KUKA KRL program: EPS_2_25748_MH01A_A_20260121065854.src

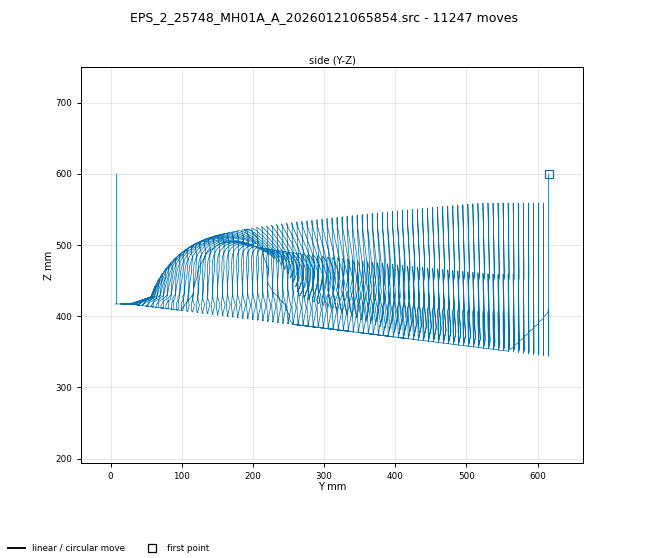
[picture p0: tool path of EPS_2_25748_MH01A_A_20260121065854.src, 11247 of 11249 moves have a stored position in this frame; points joined in program order, loops and branches not executed]
&ACCESS RVP
&REL 4
&COMMENT QRS 19112012
&PARAM EDITMASK = *
DEF PART()
EXT BAS (BAS_COMMAND :IN,REAL :IN )
INT I
BAS (#INITMOV,0 )

;KUKA QRS Post kuka4.cps  Date:22-06-2017 !

File_ID=2996

QRS_PRE_INIT()

;Init var - Until changes are made in qrs_pre_init
Outlet_Square_prg=0
Inlet_1_Square_prg=0
Inlet_2_Square_prg=0
Inlet_3_Square_prg=0
Inlet_4_Square_prg=0
Inlet_5_Square_prg=0

Outlet_1={X 0.000, Y 520.860, Z 458.500, B 0.000, E1 0.000 }
Inlet_1={X 0.000, Y 535.970, Z 408.500, B 0.000, E1 90.000 }
Outlet_1_type=201
Inlet_1_type=101
;QRS#1=Sidecore dimensions
;QRS#2=200-8" PVC SDR 35
;QRS#3=100-4" PVC SDR 28
;QRS#4=
;QRS#5=
;QRS#6=
;QRS#7=
;QRS#8=
;QRS#9=12-08 PSX
;QRS#10=8QRS PSX
;QRS#11=
;QRS#12=
;QRS#13=
;QRS#14=
;QRS#15=
;QRS#16=1220x127x838 2,75'
;QRS#17=EPS Height
;QRS#18=559
;QRS#19=*
;QRS#20= UPDATED VERSION 22-06-2017
;QRS#21=*
Outlet_Square=0100
Inlet_1_Square=045
Inlet_2_Square=0
Inlet_3_Square=0
Inlet_4_Square=0
Inlet_5_Square=0
Mill_Square=1
Outlet_Square_Prg=204
Inlet_1_Square_prg=201

QRS_INIT()

$ADVANCE=5

; T1
PTP {E1 173.434,E2 173.434}
PTP {X 0,Y 615.49,A -85,B 0,C 180,E1 173.434,E2 173.434,E3 0,E4 0,E5 0,E6 0}
QRS_SPEED_INIT()
LIN {X 0,Y 615.49,Z 600,A -85,B 0,C 180,E1 173.434,E2 173.434,E3 0,E4 0,E5 0,E6 0} C_VEL
LIN {X 0,Y 615.49,Z 432.445,A -85,B 0,C 180,E1 173.434,E2 173.434} C_VEL
LIN {X 0,Y 615.49,Z 411.751,A -85,B 0,C 180,E1 173.434,E2 173.434} C_VEL
LIN {X 0,Y 615.49,Z 411.058,A -85,B 0,C 180,E1 173.422,E2 173.422} C_VEL
LIN {X 0,Y 615.491,Z 403.195,A -85,B 0,C 180,E1 173.163,E2 173.163} C_VEL
LIN {X 0,Y 615.49,Z 396.798,A -85,B 0,C 180,E1 170.801,E2 170.801} C_VEL
LIN {X 0,Y 615.486,Z 389.623,A -85,B 0,C 180,E1 168.139,E2 168.139} C_VEL
LIN {X 0,Y 615.481,Z 382.466,A -85,B 0,C 180,E1 165.451,E2 165.451} C_VEL
LIN {X 0,Y 615.496,Z 375.278,A -85,B 0,C 180,E1 162.73,E2 162.73} C_VEL
LIN {X 0,Y 615.491,Z 368.112,A -85,B 0,C 180,E1 159.967,E2 159.967} C_VEL
LIN {X 0,Y 615.482,Z 360.924,A -85,B 0,C 180,E1 157.155,E2 157.155} C_VEL
LIN {X 0,Y 615.476,Z 354.12,A -85,B 0,C 180,E1 154.434,E2 154.434} C_VEL
LIN {X 0,Y 615.483,Z 348.349,A -85,B 0,C 180,E1 152.085,E2 152.085} C_VEL
LIN {X 0,Y 615.494,Z 343.693,A -85,B 0,C 180,E1 150.114,E2 150.114} C_VEL
LIN {X 0,Y 615.477,Z 343.693,A -85,B 0,C 180,E1 147.542,E2 147.542} C_VEL
LIN {X 0,Y 615.497,Z 343.694,A -85,B 0,C 180,E1 145.185,E2 145.185} C_VEL
LIN {X 0,Y 615.479,Z 343.69,A -85,B 0,C 180,E1 142.757,E2 142.757} C_VEL
LIN {X 0,Y 615.483,Z 343.692,A -85,B 0,C 180,E1 139.912,E2 139.912} C_VEL
LIN {X 0,Y 615.49,Z 343.699,A -85,B 0,C 180,E1 136.953,E2 136.953} C_VEL
LIN {X 0,Y 615.49,Z 343.694,A -85,B 0,C 180,E1 133.997,E2 133.997} C_VEL
LIN {X 0,Y 615.49,Z 343.689,A -85,B 0,C 180,E1 131.474,E2 131.474} C_VEL
LIN {X 0,Y 615.488,Z 343.697,A -85,B 0,C 180,E1 128.905,E2 128.905} C_VEL
LIN {X 0,Y 615.485,Z 343.69,A -85,B 0,C 180,E1 126.425,E2 126.425} C_VEL
LIN {X 0,Y 615.499,Z 343.695,A -85,B 0,C 180,E1 123.535,E2 123.535} C_VEL
LIN {X 0,Y 615.478,Z 343.692,A -85,B 0,C 180,E1 120.92,E2 120.92} C_VEL
LIN {X 0,Y 615.492,Z 343.694,A -85,B 0,C 180,E1 118.45,E2 118.45} C_VEL
LIN {X 0,Y 615.499,Z 343.694,A -85,B 0,C 180,E1 115.57,E2 115.57} C_VEL
LIN {X 0,Y 615.482,Z 343.689,A -85,B 0,C 180,E1 112.845,E2 112.845} C_VEL
LIN {X 0,Y 615.489,Z 343.693,A -85,B 0,C 180,E1 110.033,E2 110.033} C_VEL
LIN {X 0,Y 615.488,Z 343.695,A -85,B 0,C 180,E1 107.271,E2 107.271} C_VEL
LIN {X 0,Y 615.481,Z 343.69,A -85,B 0,C 180,E1 104.549,E2 104.549} C_VEL
LIN {X 0,Y 615.494,Z 343.697,A -85,B 0,C 180,E1 101.861,E2 101.861} C_VEL
LIN {X 0,Y 615.479,Z 343.692,A -85,B 0,C 180,E1 99.199,E2 99.199} C_VEL
LIN {X 0,Y 615.479,Z 343.693,A -85,B 0,C 180,E1 96.557,E2 96.557} C_VEL
LIN {X 0,Y 615.492,Z 343.694,A -85,B 0,C 180,E1 93.929,E2 93.929} C_VEL
LIN {X 0,Y 615.48,Z 343.69,A -85,B 0,C 180,E1 91.309,E2 91.309} C_VEL
LIN {X 0,Y 615.498,Z 343.7,A -85,B 0,C 180,E1 88.691,E2 88.691} C_VEL
LIN {X 0,Y 615.488,Z 343.688,A -85,B 0,C 180,E1 86.072,E2 86.072} C_VEL
LIN {X 0,Y 615.482,Z 343.697,A -85,B 0,C 180,E1 83.429,E2 83.429} C_VEL
LIN {X 0,Y 615.479,Z 343.693,A -85,B 0,C 180,E1 80.801,E2 80.801} C_VEL
LIN {X 0,Y 615.488,Z 343.69,A -85,B 0,C 180,E1 78.139,E2 78.139} C_VEL
LIN {X 0,Y 615.487,Z 343.699,A -85,B 0,C 180,E1 75.451,E2 75.451} C_VEL
LIN {X 0,Y 615.478,Z 343.691,A -85,B 0,C 180,E1 72.729,E2 72.729} C_VEL
LIN {X 0,Y 615.48,Z 343.695,A -85,B 0,C 180,E1 69.967,E2 69.967} C_VEL
LIN {X 0,Y 615.493,Z 343.696,A -85,B 0,C 180,E1 67.156,E2 67.156} C_VEL
LIN {X 0,Y 615.489,Z 343.689,A -85,B 0,C 180,E1 64.284,E2 64.284} C_VEL
LIN {X 0,Y 615.484,Z 343.69,A -85,B 0,C 180,E1 61.342,E2 61.342} C_VEL
LIN {X 0,Y 615.479,Z 343.697,A -85,B 0,C 180,E1 58.916,E2 58.916} C_VEL
LIN {X 0,Y 615.493,Z 343.69,A -85,B 0,C 180,E1 56.466,E2 56.466} C_VEL
LIN {X 0,Y 615.486,Z 343.702,A -85,B 0,C 180,E1 53.575,E2 53.575} C_VEL
LIN {X 0,Y 615.482,Z 343.69,A -85,B 0,C 180,E1 50.939,E2 50.939} C_VEL
LIN {X 0,Y 615.488,Z 343.7,A -85,B 0,C 180,E1 48.526,E2 48.526} C_VEL
LIN {X 0,Y 615.491,Z 343.689,A -85,B 0,C 180,E1 45.851,E2 45.851} C_VEL
LIN {X 0,Y 615.485,Z 343.69,A -85,B 0,C 180,E1 43.047,E2 43.047} C_VEL
LIN {X 0,Y 615.491,Z 343.693,A -85,B 0,C 180,E1 40.606,E2 40.606} C_VEL
LIN {X 0,Y 615.483,Z 343.691,A -85,B 0,C 180,E1 38.011,E2 38.011} C_VEL
LIN {X 0,Y 615.482,Z 343.694,A -85,B 0,C 180,E1 35.616,E2 35.616} C_VEL
LIN {X 0,Y 615.49,Z 343.692,A -85,B 0,C 180,E1 33.236,E2 33.236} C_VEL
LIN {X 0,Y 615.489,Z 343.688,A -85,B 0,C 180,E1 30.92,E2 30.92} C_VEL
LIN {X 0,Y 615.48,Z 343.7,A -85,B 0,C 180,E1 28.449,E2 28.449} C_VEL
LIN {X 0,Y 615.478,Z 343.693,A -85,B 0,C 180,E1 25.716,E2 25.716} C_VEL
LIN {X 0,Y 615.487,Z 343.702,A -85,B 0,C 180,E1 23.557,E2 23.557} C_VEL
LIN {X 0,Y 615.48,Z 343.692,A -85,B 0,C 180,E1 20.731,E2 20.731} C_VEL
LIN {X 0,Y 615.48,Z 343.691,A -85,B 0,C 180,E1 17.957,E2 17.957} C_VEL
LIN {X 0,Y 615.489,Z 343.702,A -85,B 0,C 180,E1 15.226,E2 15.226} C_VEL
LIN {X 0,Y 615.484,Z 343.69,A -85,B 0,C 180,E1 12.53,E2 12.53} C_VEL
LIN {X 0,Y 615.482,Z 343.694,A -85,B 0,C 180,E1 9.862,E2 9.862} C_VEL
LIN {X 0,Y 615.492,Z 343.693,A -85,B 0,C 180,E1 7.216,E2 7.216} C_VEL
LIN {X 0,Y 615.485,Z 343.69,A -85,B 0,C 180,E1 4.585,E2 4.585} C_VEL
LIN {X 0,Y 615.491,Z 343.7,A -85,B 0,C 180,E1 1.963,E2 1.963} C_VEL
LIN {X 0,Y 615.483,Z 343.689,A -85,B 0,C 180,E1 -0.654,E2 -0.654} C_VEL
LIN {X 0,Y 615.496,Z 343.696,A -85,B 0,C 180,E1 -3.273,E2 -3.273} C_VEL
LIN {X 0,Y 615.478,Z 343.692,A -85,B 0,C 180,E1 -5.899,E2 -5.899} C_VEL
LIN {X 0,Y 615.483,Z 343.693,A -85,B 0,C 180,E1 -8.537,E2 -8.537} C_VEL
LIN {X 0,Y 615.486,Z 343.695,A -85,B 0,C 180,E1 -11.193,E2 -11.193} C_VEL
LIN {X 0,Y 615.478,Z 343.69,A -85,B 0,C 180,E1 -13.928,E2 -13.928} C_VEL
LIN {X 0,Y 615.484,Z 343.7,A -85,B 0,C 180,E1 -16.587,E2 -16.587} C_VEL
LIN {X 0,Y 615.488,Z 343.691,A -85,B 0,C 180,E1 -19.338,E2 -19.338} C_VEL
LIN {X 0,Y 615.494,Z 343.687,A -85,B 0,C 180,E1 -22.136,E2 -22.136} C_VEL
LIN {X 0,Y 615.497,Z 343.695,A -85,B 0,C 180,E1 -24.991,E2 -24.991} C_VEL
LIN {X 0,Y 615.489,Z 343.688,A -85,B 0,C 180,E1 -27.177,E2 -27.177} C_VEL
LIN {X 0,Y 615.488,Z 343.693,A -85,B 0,C 180,E1 -30.16,E2 -30.16} C_VEL
LIN {X 0,Y 615.477,Z 343.691,A -85,B 0,C 180,E1 -32.458,E2 -32.458} C_VEL
LIN {X 0,Y 615.498,Z 343.7,A -85,B 0,C 180,E1 -34.815,E2 -34.815} C_VEL
LIN {X 0,Y 615.479,Z 343.69,A -85,B 0,C 180,E1 -37.243,E2 -37.243} C_VEL
LIN {X 0,Y 615.482,Z 343.696,A -85,B 0,C 180,E1 -40.088,E2 -40.088} C_VEL
LIN {X 0,Y 615.477,Z 343.69,A -85,B 0,C 180,E1 -42.354,E2 -42.354} C_VEL
LIN {X 0,Y 615.485,Z 343.696,A -85,B 0,C 180,E1 -45.069,E2 -45.069} C_VEL
LIN {X 0,Y 615.492,Z 343.694,A -85,B 0,C 180,E1 -47.92,E2 -47.92} C_VEL
LIN {X 0,Y 615.48,Z 343.694,A -85,B 0,C 180,E1 -50.249,E2 -50.249} C_VEL
LIN {X 0,Y 615.484,Z 343.7,A -85,B 0,C 180,E1 -53.064,E2 -53.064} C_VEL
LIN {X 0,Y 615.488,Z 343.691,A -85,B 0,C 180,E1 -55.3,E2 -55.3} C_VEL
LIN {X 0,Y 615.494,Z 343.689,A -85,B 0,C 180,E1 -57.669,E2 -57.669} C_VEL
LIN {X 0,Y 615.492,Z 343.687,A -85,B 0,C 180,E1 -60.594,E2 -60.594} C_VEL
LIN {X 0,Y 615.485,Z 343.84,A -85,B 0,C 180,E1 -62.593,E2 -62.593} C_VEL
LIN {X 0,Y 615.489,Z 361.437,A -85,B 0,C 180,E1 -65.369,E2 -65.369} C_VEL
LIN {X 0,Y 615.488,Z 379.893,A -85,B 0,C 180,E1 -68.216,E2 -68.216} C_VEL
LIN {X 0,Y 615.492,Z 398.328,A -85,B 0,C 180,E1 -71.009,E2 -71.009} C_VEL
LIN {X 0,Y 615.493,Z 417.271,A -85,B 0,C 180,E1 -73.832,E2 -73.832} C_VEL
LIN {X 0,Y 615.478,Z 436.291,A -85,B 0,C 180,E1 -76.631,E2 -76.631} C_VEL
LIN {X 0,Y 615.497,Z 447.778,A -85,B 0,C 180,E1 -78.306,E2 -78.306} C_VEL
LIN {X 0,Y 615.483,Z 462.241,A -85,B 0,C 180,E1 -78.557,E2 -78.557} C_VEL
LIN {X 0,Y 615.481,Z 475.314,A -85,B 0,C 180,E1 -78.921,E2 -78.921} C_VEL
LIN {X 0,Y 615.489,Z 487.118,A -85,B 0,C 180,E1 -79.383,E2 -79.383} C_VEL
LIN {X 0,Y 615.487,Z 498.575,A -85,B 0,C 180,E1 -79.972,E2 -79.972} C_VEL
LIN {X 0,Y 615.499,Z 510.021,A -85,B 0,C 180,E1 -80.719,E2 -80.719} C_VEL
LIN {X 0,Y 615.498,Z 519.257,A -85,B 0,C 180,E1 -81.464,E2 -81.464} C_VEL
LIN {X 0,Y 615.499,Z 527.654,A -85,B 0,C 180,E1 -82.29,E2 -82.29} C_VEL
LIN {X 0,Y 615.497,Z 535.69,A -85,B 0,C 180,E1 -83.259,E2 -83.259} C_VEL
LIN {X 0,Y 615.499,Z 541.423,A -85,B 0,C 180,E1 -84.102,E2 -84.102} C_VEL
LIN {X 0,Y 615.496,Z 546.873,A -85,B 0,C 180,E1 -85.087,E2 -85.087} C_VEL
LIN {X 0,Y 615.496,Z 551.141,A -85,B 0,C 180,E1 -86.072,E2 -86.072} C_VEL
LIN {X 0,Y 615.495,Z 553.399,A -85,B 0,C 180,E1 -86.727,E2 -86.727} C_VEL
LIN {X 0,Y 615.497,Z 555.233,A -85,B 0,C 180,E1 -87.382,E2 -87.382} C_VEL
LIN {X 0,Y 615.499,Z 556.608,A -85,B 0,C 180,E1 -88.037,E2 -88.037} C_VEL
LIN {X 0,Y 615.496,Z 558.174,A -85,B 0,C 180,E1 -89.346,E2 -89.346} C_VEL
LIN {X 0,Y 615.494,Z 558.389,A -85,B 0,C 180,E1 -90,E2 -90} C_VEL
LIN {X 0,Y 615.496,Z 557.58,A -85,B 0,C 180,E1 -91.309,E2 -91.309} C_VEL
LIN {X 0,Y 615.499,Z 556.607,A -85,B 0,C 180,E1 -91.963,E2 -91.963} C_VEL
LIN {X 0,Y 615.497,Z 555.233,A -85,B 0,C 180,E1 -92.618,E2 -92.618} C_VEL
LIN {X 0,Y 615.496,Z 552.349,A -85,B 0,C 180,E1 -93.601,E2 -93.601} C_VEL
LIN {X 0,Y 615.498,Z 548.441,A -85,B 0,C 180,E1 -94.585,E2 -94.585} C_VEL
LIN {X 0,Y 615.499,Z 543.404,A -85,B 0,C 180,E1 -95.57,E2 -95.57} C_VEL
LIN {X 0,Y 615.497,Z 536.869,A -85,B 0,C 180,E1 -96.583,E2 -96.583} C_VEL
LIN {X 0,Y 615.497,Z 529.132,A -85,B 0,C 180,E1 -97.545,E2 -97.545} C_VEL
LIN {X 0,Y 615.498,Z 521.044,A -85,B 0,C 180,E1 -98.371,E2 -98.371} C_VEL
LIN {X 0,Y 615.499,Z 511.166,A -85,B 0,C 180,E1 -99.199,E2 -99.199} C_VEL
LIN {X 0,Y 615.492,Z 499.979,A -85,B 0,C 180,E1 -99.945,E2 -99.945} C_VEL
LIN {X 0,Y 615.484,Z 489.021,A -85,B 0,C 180,E1 -100.527,E2 -100.527} C_VEL
LIN {X 0,Y 615.482,Z 476.474,A -85,B 0,C 180,E1 -101.041,E2 -101.041} C_VEL
LIN {X 0,Y 615.481,Z 464.062,A -85,B 0,C 180,E1 -101.402,E2 -101.402} C_VEL
LIN {X 0,Y 615.495,Z 450.456,A -85,B 0,C 180,E1 -101.652,E2 -101.652} C_VEL
LIN {X 0,Y 615.497,Z 447.777,A -85,B 0,C 180,E1 -101.694,E2 -101.694} C_VEL
LIN {X 0,Y 615.494,Z 427.093,A -85,B 0,C 180,E1 -104.718,E2 -104.718} C_VEL
LIN {X 0,Y 615.492,Z 407.537,A -85,B 0,C 180,E1 -107.613,E2 -107.613} C_VEL
LIN {X 0,Y 615.487,Z 389.681,A -85,B 0,C 180,E1 -110.295,E2 -110.295} C_VEL
LIN {X 0,Y 615.479,Z 371.82,A -85,B 0,C 180,E1 -113.023,E2 -113.023} C_VEL
LIN {X 0,Y 615.5,Z 354.513,A -85,B 0,C 180,E1 -115.715,E2 -115.715} C_VEL
LIN {X 0,Y 615.49,Z 343.697,A -85,B 0,C 180,E1 -117.453,E2 -117.453} C_VEL
LIN {X 0,Y 615.494,Z 343.698,A -85,B 0,C 180,E1 -120.16,E2 -120.16} C_VEL
LIN {X 0,Y 615.495,Z 343.696,A -85,B 0,C 180,E1 -122.457,E2 -122.457} C_VEL
LIN {X 0,Y 615.485,Z 343.698,A -85,B 0,C 180,E1 -124.815,E2 -124.815} C_VEL
LIN {X 0,Y 615.487,Z 343.701,A -85,B 0,C 180,E1 -127.242,E2 -127.242} C_VEL
LIN {X 0,Y 615.485,Z 343.698,A -85,B 0,C 180,E1 -130.088,E2 -130.088} C_VEL
LIN {X 0,Y 615.499,Z 343.696,A -85,B 0,C 180,E1 -132.352,E2 -132.352} C_VEL
LIN {X 0,Y 615.48,Z 343.699,A -85,B 0,C 180,E1 -135.07,E2 -135.07} C_VEL
LIN {X 0,Y 615.498,Z 343.7,A -85,B 0,C 180,E1 -137.919,E2 -137.919} C_VEL
LIN {X 0,Y 615.492,Z 343.697,A -85,B 0,C 180,E1 -140.25,E2 -140.25} C_VEL
LIN {X 0,Y 615.485,Z 343.702,A -85,B 0,C 180,E1 -143.064,E2 -143.064} C_VEL
LIN {X 0,Y 615.491,Z 343.697,A -85,B 0,C 180,E1 -145.978,E2 -145.978} C_VEL
LIN {X 0,Y 615.496,Z 343.699,A -85,B 0,C 180,E1 -148.315,E2 -148.315} C_VEL
LIN {X 0,Y 615.491,Z 343.791,A -85,B 0,C 180,E1 -150.303,E2 -150.303} C_VEL
LIN {X 0,Y 615.498,Z 350.25,A -85,B 0,C 180,E1 -152.954,E2 -152.954} C_VEL
LIN {X 0,Y 615.489,Z 357.77,A -85,B 0,C 180,E1 -155.992,E2 -155.992} C_VEL
LIN {X 0,Y 615.478,Z 364.291,A -85,B 0,C 180,E1 -158.568,E2 -158.568} C_VEL
LIN {X 0,Y 615.477,Z 371.461,A -85,B 0,C 180,E1 -161.354,E2 -161.354} C_VEL
LIN {X 0,Y 615.492,Z 378.634,A -85,B 0,C 180,E1 -164.095,E2 -164.095} C_VEL
LIN {X 0,Y 615.494,Z 385.799,A -85,B 0,C 180,E1 -166.799,E2 -166.799} C_VEL
LIN {X 0,Y 615.486,Z 392.972,A -85,B 0,C 180,E1 -169.473,E2 -169.473} C_VEL
LIN {X 0,Y 615.477,Z 400.129,A -85,B 0,C 180,E1 -172.124,E2 -172.124} C_VEL
LIN {X 0,Y 615.484,Z 403.219,A -85,B 0,C 180,E1 -173.261,E2 -173.261} C_VEL
LIN {X 0,Y 615.493,Z 413.526,A -85,B 0,C 180,E1 -173.608,E2 -173.608} C_VEL
LIN {X 0,Y 615.478,Z 421.946,A -85,B 0,C 180,E1 -174.019,E2 -174.019} C_VEL
LIN {X 0,Y 615.486,Z 429.671,A -85,B 0,C 180,E1 -174.512,E2 -174.512} C_VEL
LIN {X 0,Y 615.481,Z 436.518,A -85,B 0,C 180,E1 -175.087,E2 -175.087} C_VEL
LIN {X 0,Y 615.497,Z 442.668,A -85,B 0,C 180,E1 -175.744,E2 -175.744} C_VEL
LIN {X 0,Y 615.497,Z 447.515,A -85,B 0,C 180,E1 -176.399,E2 -176.399} C_VEL
LIN {X 0,Y 615.496,Z 451.25,A -85,B 0,C 180,E1 -177.055,E2 -177.055} C_VEL
LIN {X 0,Y 615.498,Z 455.23,A -85,B 0,C 180,E1 -178.037,E2 -178.037} C_VEL
LIN {X 0,Y 615.495,Z 456.964,A -85,B 0,C 180,E1 -178.691,E2 -178.691} C_VEL
LIN {X 0,Y 615.497,Z 458.004,A -85,B 0,C 180,E1 -179.346,E2 -179.346} C_VEL
LIN {X 0,Y 615.494,Z 458.384,A -85,B 0,C 180,E1 -180,E2 -180} C_VEL
LIN {X 0,Y 615.496,Z 458.105,A -85,B 0,C 180,E1 -180.654,E2 -180.654} C_VEL
LIN {X 0,Y 615.498,Z 457.165,A -85,B 0,C 180,E1 -181.309,E2 -181.309} C_VEL
LIN {X 0,Y 615.496,Z 455.536,A -85,B 0,C 180,E1 -181.963,E2 -181.963} C_VEL
LIN {X 0,Y 615.498,Z 451.663,A -85,B 0,C 180,E1 -182.945,E2 -182.945} C_VEL
LIN {X 0,Y 615.5,Z 447.011,A -85,B 0,C 180,E1 -183.765,E2 -183.765} C_VEL
LIN {X 0,Y 615.499,Z 442.03,A -85,B 0,C 180,E1 -184.42,E2 -184.42} C_VEL
LIN {X 0,Y 615.492,Z 435.752,A -85,B 0,C 180,E1 -185.077,E2 -185.077} C_VEL
LIN {X 0,Y 615.483,Z 428.588,A -85,B 0,C 180,E1 -185.652,E2 -185.652} C_VEL
LIN {X 0,Y 615.483,Z 420.604,A -85,B 0,C 180,E1 -186.145,E2 -186.145} C_VEL
LIN {X 0,Y 615.49,Z 411.058,A -85,B 0,C 180,E1 -186.578,E2 -186.578} C_VEL
LIN {X 0,Y 615.134,Z 407.804,A -85,B 0,C 180,E1 -186.754,E2 -186.754} C_VEL
LIN {X 0,Y 614.28,Z 405.203,A -85,B 0,C 180,E1 -187.003,E2 -187.003} C_VEL
LIN {X 0,Y 612.526,Z 402.365,A -85,B 0,C 180,E1 -187.458,E2 -187.458} C_VEL
LIN {X 0,Y 610.614,Z 400.714,A -85,B 0,C 180,E1 -187.986,E2 -187.986} C_VEL
LIN {X 0,Y 608.705,Z 398.756,A -85,B 0,C 180,E1 -188.746,E2 -188.746} C_VEL
LIN {X 0,Y 608.412,Z 397.698,A -85,B 0,C 180,E1 -189.134,E2 -189.134} C_VEL
LIN {X 0,Y 608.424,Z 390.014,A -85,B 0,C 180,E1 -192.001,E2 -192.001} C_VEL
LIN {X 0,Y 608.441,Z 382.795,A -85,B 0,C 180,E1 -194.721,E2 -194.721} C_VEL
LIN {X 0,Y 608.459,Z 375.575,A -85,B 0,C 180,E1 -197.477,E2 -197.477} C_VEL
LIN {X 0,Y 608.443,Z 368.356,A -85,B 0,C 180,E1 -200.275,E2 -200.275} C_VEL
LIN {X 0,Y 608.446,Z 361.136,A -85,B 0,C 180,E1 -203.124,E2 -203.124} C_VEL
LIN {X 0,Y 608.465,Z 354.69,A -85,B 0,C 180,E1 -205.719,E2 -205.719} C_VEL
LIN {X 0,Y 608.476,Z 347.645,A -85,B 0,C 180,E1 -208.62,E2 -208.62} C_VEL
LIN {X 0,Y 608.481,Z 344.69,A -85,B 0,C 180,E1 -209.905,E2 -209.905} C_VEL
LIN {X 0,Y 608.454,Z 344.692,A -85,B 0,C 180,E1 -212.521,E2 -212.521} C_VEL
LIN {X 0,Y 608.444,Z 344.692,A -85,B 0,C 180,E1 -215.278,E2 -215.278} C_VEL
LIN {X 0,Y 608.468,Z 344.693,A -85,B 0,C 180,E1 -217.747,E2 -217.747} C_VEL
LIN {X 0,Y 608.448,Z 344.691,A -85,B 0,C 180,E1 -220.328,E2 -220.328} C_VEL
LIN {X 0,Y 608.455,Z 344.698,A -85,B 0,C 180,E1 -222.96,E2 -222.96} C_VEL
LIN {X 0,Y 608.461,Z 344.69,A -85,B 0,C 180,E1 -225.736,E2 -225.736} C_VEL
LIN {X 0,Y 608.464,Z 344.689,A -85,B 0,C 180,E1 -228.658,E2 -228.658} C_VEL
LIN {X 0,Y 608.465,Z 344.69,A -85,B 0,C 180,E1 -231.76,E2 -231.76} C_VEL
LIN {X 0,Y 608.448,Z 344.691,A -85,B 0,C 180,E1 -233.955,E2 -233.955} C_VEL
LIN {X 0,Y 608.47,Z 344.696,A -85,B 0,C 180,E1 -236.329,E2 -236.329} C_VEL
LIN {X 0,Y 608.449,Z 344.691,A -85,B 0,C 180,E1 -238.733,E2 -238.733} C_VEL
LIN {X 0,Y 608.479,Z 344.694,A -85,B 0,C 180,E1 -241.38,E2 -241.38} C_VEL
LIN {X 0,Y 608.446,Z 344.692,A -85,B 0,C 180,E1 -243.964,E2 -243.964} C_VEL
LIN {X 0,Y 608.465,Z 344.694,A -85,B 0,C 180,E1 -246.155,E2 -246.155} C_VEL
LIN {X 0,Y 608.47,Z 344.691,A -85,B 0,C 180,E1 -248.308,E2 -248.308} C_VEL
LIN {X 0,Y 608.457,Z 344.695,A -85,B 0,C 180,E1 -251.13,E2 -251.13} C_VEL
LIN {X 0,Y 608.459,Z 344.69,A -85,B 0,C 180,E1 -253.906,E2 -253.906} C_VEL
LIN {X 0,Y 608.46,Z 344.693,A -85,B 0,C 180,E1 -256.643,E2 -256.643} C_VEL
LIN {X 0,Y 608.466,Z 344.692,A -85,B 0,C 180,E1 -259.35,E2 -259.35} C_VEL
LIN {X 0,Y 608.481,Z 344.687,A -85,B 0,C 180,E1 -262.033,E2 -262.033} C_VEL
LIN {X 0,Y 608.472,Z 344.695,A -85,B 0,C 180,E1 -264.698,E2 -264.698} C_VEL
LIN {X 0,Y 608.472,Z 344.688,A -85,B 0,C 180,E1 -267.352,E2 -267.352} C_VEL
LIN {X 0,Y 608.482,Z 344.69,A -85,B 0,C 180,E1 -270,E2 -270} C_VEL
LIN {X 0,Y 608.472,Z 344.691,A -85,B 0,C 180,E1 -272.648,E2 -272.648} C_VEL
LIN {X 0,Y 608.462,Z 344.69,A -85,B 0,C 180,E1 -275.302,E2 -275.302} C_VEL
LIN {X 0,Y 608.482,Z 344.694,A -85,B 0,C 180,E1 -277.967,E2 -277.967} C_VEL
LIN {X 0,Y 608.47,Z 344.691,A -85,B 0,C 180,E1 -280.954,E2 -280.954} C_VEL
LIN {X 0,Y 608.465,Z 344.692,A -85,B 0,C 180,E1 -283.356,E2 -283.356} C_VEL
LIN {X 0,Y 608.468,Z 344.692,A -85,B 0,C 180,E1 -286.094,E2 -286.094} C_VEL
LIN {X 0,Y 608.457,Z 344.69,A -85,B 0,C 180,E1 -288.87,E2 -288.87} C_VEL
LIN {X 0,Y 608.472,Z 344.691,A -85,B 0,C 180,E1 -291.691,E2 -291.691} C_VEL
LIN {X 0,Y 608.451,Z 344.697,A -85,B 0,C 180,E1 -294.571,E2 -294.571} C_VEL
LIN {X 0,Y 608.472,Z 344.688,A -85,B 0,C 180,E1 -297.205,E2 -297.205} C_VEL
LIN {X 0,Y 608.465,Z 344.693,A -85,B 0,C 180,E1 -299.971,E2 -299.971} C_VEL
LIN {X 0,Y 608.464,Z 344.694,A -85,B 0,C 180,E1 -302.879,E2 -302.879} C_VEL
LIN {X 0,Y 608.446,Z 344.692,A -85,B 0,C 180,E1 -305.278,E2 -305.278} C_VEL
LIN {X 0,Y 608.472,Z 344.693,A -85,B 0,C 180,E1 -308.24,E2 -308.24} C_VEL
LIN {X 0,Y 608.447,Z 344.692,A -85,B 0,C 180,E1 -310.328,E2 -310.328} C_VEL
LIN {X 0,Y 608.485,Z 344.69,A -85,B 0,C 180,E1 -313.31,E2 -313.31} C_VEL
LIN {X 0,Y 608.469,Z 344.692,A -85,B 0,C 180,E1 -316.13,E2 -316.13} C_VEL
LIN {X 0,Y 608.451,Z 344.691,A -85,B 0,C 180,E1 -318.823,E2 -318.823} C_VEL
LIN {X 0,Y 608.465,Z 344.691,A -85,B 0,C 180,E1 -321.76,E2 -321.76} C_VEL
LIN {X 0,Y 608.451,Z 344.691,A -85,B 0,C 180,E1 -323.954,E2 -323.954} C_VEL
LIN {X 0,Y 608.471,Z 344.695,A -85,B 0,C 180,E1 -326.329,E2 -326.329} C_VEL
LIN {X 0,Y 608.449,Z 344.691,A -85,B 0,C 180,E1 -328.732,E2 -328.732} C_VEL
LIN {X 0,Y 608.472,Z 344.695,A -85,B 0,C 180,E1 -331.381,E2 -331.381} C_VEL
LIN {X 0,Y 608.437,Z 344.692,A -85,B 0,C 180,E1 -333.964,E2 -333.964} C_VEL
LIN {X 0,Y 608.471,Z 344.692,A -85,B 0,C 180,E1 -336.155,E2 -336.155} C_VEL
LIN {X 0,Y 608.454,Z 344.69,A -85,B 0,C 180,E1 -339.018,E2 -339.018} C_VEL
LIN {X 0,Y 608.448,Z 344.693,A -85,B 0,C 180,E1 -341.828,E2 -341.828} C_VEL
LIN {X 0,Y 608.471,Z 344.693,A -85,B 0,C 180,E1 -344.594,E2 -344.594} C_VEL
LIN {X 0,Y 608.476,Z 344.688,A -85,B 0,C 180,E1 -347.323,E2 -347.323} C_VEL
LIN {X 0,Y 608.453,Z 344.694,A -85,B 0,C 180,E1 -350.023,E2 -350.023} C_VEL
LIN {X 0,Y 608.469,Z 344.691,A -85,B 0,C 180,E1 -352.701,E2 -352.701} C_VEL
LIN {X 0,Y 608.455,Z 344.691,A -85,B 0,C 180,E1 -355.362,E2 -355.362} C_VEL
LIN {X 0,Y 608.46,Z 344.696,A -85,B 0,C 180,E1 -358.014,E2 -358.014} C_VEL
LIN {X 0,Y 608.478,Z 344.687,A -85,B 0,C 180,E1 -360.662,E2 -360.662} C_VEL
LIN {X 0,Y 608.488,Z 344.691,A -85,B 0,C 180,E1 -363.311,E2 -363.311} C_VEL
LIN {X 0,Y 608.453,Z 344.692,A -85,B 0,C 180,E1 -365.967,E2 -365.967} C_VEL
LIN {X 0,Y 608.455,Z 344.691,A -85,B 0,C 180,E1 -368.636,E2 -368.636} C_VEL
LIN {X 0,Y 608.477,Z 344.693,A -85,B 0,C 180,E1 -371.324,E2 -371.324} C_VEL
LIN {X 0,Y 608.471,Z 344.688,A -85,B 0,C 180,E1 -374.037,E2 -374.037} C_VEL
LIN {X 0,Y 608.477,Z 344.69,A -85,B 0,C 180,E1 -376.783,E2 -376.783} C_VEL
LIN {X 0,Y 608.457,Z 344.694,A -85,B 0,C 180,E1 -379.57,E2 -379.57} C_VEL
LIN {X 0,Y 608.462,Z 344.69,A -85,B 0,C 180,E1 -382.476,E2 -382.476} C_VEL
LIN {X 0,Y 608.46,Z 344.694,A -85,B 0,C 180,E1 -384.571,E2 -384.571} C_VEL
LIN {X 0,Y 608.452,Z 344.691,A -85,B 0,C 180,E1 -387.518,E2 -387.518} C_VEL
LIN {X 0,Y 608.475,Z 344.693,A -85,B 0,C 180,E1 -389.972,E2 -389.972} C_VEL
LIN {X 0,Y 608.457,Z 344.694,A -85,B 0,C 180,E1 -392.88,E2 -392.88} C_VEL
LIN {X 0,Y 608.445,Z 344.693,A -85,B 0,C 180,E1 -395.278,E2 -395.278} C_VEL
LIN {X 0,Y 608.476,Z 344.694,A -85,B 0,C 180,E1 -398.241,E2 -398.241} C_VEL
LIN {X 0,Y 608.453,Z 344.693,A -85,B 0,C 180,E1 -401.177,E2 -401.177} C_VEL
LIN {X 0,Y 608.47,Z 344.688,A -85,B 0,C 180,E1 -403.87,E2 -403.87} C_VEL
LIN {X 0,Y 608.483,Z 344.691,A -85,B 0,C 180,E1 -406.69,E2 -406.69} C_VEL
LIN {X 0,Y 608.455,Z 344.691,A -85,B 0,C 180,E1 -408.823,E2 -408.823} C_VEL
LIN {X 0,Y 608.464,Z 344.693,A -85,B 0,C 180,E1 -411.76,E2 -411.76} C_VEL
LIN {X 0,Y 608.447,Z 344.691,A -85,B 0,C 180,E1 -413.955,E2 -413.955} C_VEL
LIN {X 0,Y 608.468,Z 344.693,A -85,B 0,C 180,E1 -416.329,E2 -416.329} C_VEL
LIN {X 0,Y 608.448,Z 344.692,A -85,B 0,C 180,E1 -418.733,E2 -418.733} C_VEL
LIN {X 0,Y 608.474,Z 344.694,A -85,B 0,C 180,E1 -421.38,E2 -421.38} C_VEL
LIN {X 0,Y 608.479,Z 344.706,A -85,B 0,C 180,E1 -422.39,E2 -422.39} C_VEL
LIN {X 0,Y 608.617,Z 357.707,A -85,B 0,C 180,E1 -424.481,E2 -424.481} C_VEL
LIN {X 0,Y 608.571,Z 375.515,A -85,B 0,C 180,E1 -427.276,E2 -427.276} C_VEL
LIN {X 0,Y 608.516,Z 393.747,A -85,B 0,C 180,E1 -430.08,E2 -430.08} C_VEL
LIN {X 0,Y 608.5,Z 411.056,A -85,B 0,C 180,E1 -432.698,E2 -432.698} C_VEL
LIN {X 0,Y 608.47,Z 429.518,A -85,B 0,C 180,E1 -435.45,E2 -435.45} C_VEL
LIN {X 0,Y 608.486,Z 447.981,A -85,B 0,C 180,E1 -438.17,E2 -438.17} C_VEL
LIN {X 0,Y 608.545,Z 463.267,A -85,B 0,C 180,E1 -438.445,E2 -438.445} C_VEL
LIN {X 0,Y 608.523,Z 475.887,A -85,B 0,C 180,E1 -438.808,E2 -438.808} C_VEL
LIN {X 0,Y 608.519,Z 487.581,A -85,B 0,C 180,E1 -439.275,E2 -439.275} C_VEL
LIN {X 0,Y 608.492,Z 498.755,A -85,B 0,C 180,E1 -439.855,E2 -439.855} C_VEL
LIN {X 0,Y 608.504,Z 510.252,A -85,B 0,C 180,E1 -440.611,E2 -440.611} C_VEL
LIN {X 0,Y 608.472,Z 519.536,A -85,B 0,C 180,E1 -441.364,E2 -441.364} C_VEL
LIN {X 0,Y 608.456,Z 527.989,A -85,B 0,C 180,E1 -442.2,E2 -442.2} C_VEL
LIN {X 0,Y 608.462,Z 536.235,A -85,B 0,C 180,E1 -443.201,E2 -443.201} C_VEL
LIN {X 0,Y 608.437,Z 542.877,A -85,B 0,C 180,E1 -444.199,E2 -444.199} C_VEL
LIN {X 0,Y 608.432,Z 548.95,A -85,B 0,C 180,E1 -445.362,E2 -445.362} C_VEL
LIN {X 0,Y 608.449,Z 552.896,A -85,B 0,C 180,E1 -446.358,E2 -446.358} C_VEL
LIN {X 0,Y 608.425,Z 555.809,A -85,B 0,C 180,E1 -447.352,E2 -447.352} C_VEL
LIN {X 0,Y 608.444,Z 557.201,A -85,B 0,C 180,E1 -448.014,E2 -448.014} C_VEL
LIN {X 0,Y 608.438,Z 558.783,A -85,B 0,C 180,E1 -449.338,E2 -449.338} C_VEL
LIN {X 0,Y 608.434,Z 559,A -85,B 0,C 180,E1 -450,E2 -450} C_VEL
LIN {X 0,Y 608.448,Z 558.184,A -85,B 0,C 180,E1 -451.324,E2 -451.324} C_VEL
LIN {X 0,Y 608.444,Z 557.201,A -85,B 0,C 180,E1 -451.986,E2 -451.986} C_VEL
LIN {X 0,Y 608.425,Z 555.809,A -85,B 0,C 180,E1 -452.648,E2 -452.648} C_VEL
LIN {X 0,Y 608.449,Z 552.896,A -85,B 0,C 180,E1 -453.642,E2 -453.642} C_VEL
LIN {X 0,Y 608.432,Z 548.95,A -85,B 0,C 180,E1 -454.638,E2 -454.638} C_VEL
LIN {X 0,Y 608.437,Z 542.876,A -85,B 0,C 180,E1 -455.801,E2 -455.801} C_VEL
LIN {X 0,Y 608.462,Z 536.234,A -85,B 0,C 180,E1 -456.799,E2 -456.799} C_VEL
LIN {X 0,Y 608.456,Z 527.988,A -85,B 0,C 180,E1 -457.8,E2 -457.8} C_VEL
LIN {X 0,Y 608.472,Z 519.535,A -85,B 0,C 180,E1 -458.636,E2 -458.636} C_VEL
LIN {X 0,Y 608.481,Z 509.089,A -85,B 0,C 180,E1 -459.473,E2 -459.473} C_VEL
LIN {X 0,Y 608.492,Z 498.754,A -85,B 0,C 180,E1 -460.145,E2 -460.145} C_VEL
LIN {X 0,Y 608.521,Z 487.26,A -85,B 0,C 180,E1 -460.74,E2 -460.74} C_VEL
LIN {X 0,Y 608.529,Z 474.882,A -85,B 0,C 180,E1 -461.225,E2 -461.225} C_VEL
LIN {X 0,Y 608.546,Z 461.434,A -85,B 0,C 180,E1 -461.597,E2 -461.597} C_VEL
LIN {X 0,Y 608.486,Z 447.98,A -85,B 0,C 180,E1 -461.83,E2 -461.83} C_VEL
LIN {X 0,Y 608.49,Z 428.364,A -85,B 0,C 180,E1 -464.72,E2 -464.72} C_VEL
LIN {X 0,Y 608.502,Z 409.901,A -85,B 0,C 180,E1 -467.475,E2 -467.475} C_VEL
LIN {X 0,Y 608.531,Z 392.592,A -85,B 0,C 180,E1 -470.096,E2 -470.096} C_VEL
LIN {X 0,Y 608.572,Z 374.131,A -85,B 0,C 180,E1 -472.939,E2 -472.939} C_VEL
LIN {X 0,Y 608.614,Z 356.269,A -85,B 0,C 180,E1 -475.748,E2 -475.748} C_VEL
LIN {X 0,Y 608.483,Z 344.705,A -85,B 0,C 180,E1 -477.61,E2 -477.61} C_VEL
LIN {X 0,Y 608.477,Z 344.692,A -85,B 0,C 180,E1 -480.545,E2 -480.545} C_VEL
LIN {X 0,Y 608.465,Z 344.695,A -85,B 0,C 180,E1 -482.879,E2 -482.879} C_VEL
LIN {X 0,Y 608.443,Z 344.699,A -85,B 0,C 180,E1 -485.278,E2 -485.278} C_VEL
LIN {X 0,Y 608.466,Z 344.694,A -85,B 0,C 180,E1 -487.747,E2 -487.747} C_VEL
LIN {X 0,Y 608.453,Z 344.697,A -85,B 0,C 180,E1 -490.329,E2 -490.329} C_VEL
LIN {X 0,Y 608.483,Z 344.692,A -85,B 0,C 180,E1 -493.31,E2 -493.31} C_VEL
LIN {X 0,Y 608.479,Z 344.692,A -85,B 0,C 180,E1 -496.131,E2 -496.131} C_VEL
LIN {X 0,Y 608.457,Z 344.697,A -85,B 0,C 180,E1 -498.823,E2 -498.823} C_VEL
LIN {X 0,Y 608.474,Z 344.693,A -85,B 0,C 180,E1 -501.412,E2 -501.412} C_VEL
LIN {X 0,Y 608.465,Z 344.695,A -85,B 0,C 180,E1 -503.953,E2 -503.953} C_VEL
LIN {X 0,Y 608.469,Z 344.696,A -85,B 0,C 180,E1 -506.33,E2 -506.33} C_VEL
LIN {X 0,Y 608.45,Z 344.696,A -85,B 0,C 180,E1 -508.732,E2 -508.732} C_VEL
LIN {X 0,Y 608.483,Z 344.805,A -85,B 0,C 180,E1 -510.316,E2 -510.316} C_VEL
LIN {X 0,Y 608.451,Z 351.891,A -85,B 0,C 180,E1 -513.226,E2 -513.226} C_VEL
LIN {X 0,Y 608.458,Z 358.354,A -85,B 0,C 180,E1 -515.852,E2 -515.852} C_VEL
LIN {X 0,Y 608.443,Z 364.518,A -85,B 0,C 180,E1 -518.307,E2 -518.307} C_VEL
LIN {X 0,Y 608.432,Z 371.734,A -85,B 0,C 180,E1 -521.13,E2 -521.13} C_VEL
LIN {X 0,Y 608.448,Z 378.95,A -85,B 0,C 180,E1 -523.906,E2 -523.906} C_VEL
LIN {X 0,Y 608.437,Z 386.166,A -85,B 0,C 180,E1 -526.643,E2 -526.643} C_VEL
LIN {X 0,Y 608.424,Z 393.383,A -85,B 0,C 180,E1 -529.349,E2 -529.349} C_VEL
LIN {X 0,Y 608.412,Z 400.599,A -85,B 0,C 180,E1 -532.032,E2 -532.032} C_VEL
LIN {X 0,Y 608.446,Z 403.882,A -85,B 0,C 180,E1 -533.187,E2 -533.187} C_VEL
LIN {X 0,Y 608.478,Z 414.08,A -85,B 0,C 180,E1 -533.534,E2 -533.534} C_VEL
LIN {X 0,Y 608.454,Z 422.473,A -85,B 0,C 180,E1 -533.95,E2 -533.95} C_VEL
LIN {X 0,Y 608.451,Z 431.253,A -85,B 0,C 180,E1 -534.532,E2 -534.532} C_VEL
LIN {X 0,Y 608.44,Z 437.028,A -85,B 0,C 180,E1 -535.03,E2 -535.03} C_VEL
LIN {X 0,Y 608.443,Z 443.206,A -85,B 0,C 180,E1 -535.694,E2 -535.694} C_VEL
LIN {X 0,Y 608.451,Z 448.068,A -85,B 0,C 180,E1 -536.358,E2 -536.358} C_VEL
LIN {X 0,Y 608.451,Z 451.818,A -85,B 0,C 180,E1 -537.021,E2 -537.021} C_VEL
LIN {X 0,Y 608.443,Z 455.825,A -85,B 0,C 180,E1 -538.014,E2 -538.014} C_VEL
LIN {X 0,Y 608.448,Z 457.569,A -85,B 0,C 180,E1 -538.676,E2 -538.676} C_VEL
LIN {X 0,Y 608.44,Z 458.615,A -85,B 0,C 180,E1 -539.338,E2 -539.338} C_VEL
LIN {X 0,Y 608.434,Z 458.995,A -85,B 0,C 180,E1 -540,E2 -540} C_VEL
LIN {X 0,Y 608.438,Z 458.714,A -85,B 0,C 180,E1 -540.662,E2 -540.662} C_VEL
LIN {X 0,Y 608.45,Z 457.768,A -85,B 0,C 180,E1 -541.324,E2 -541.324} C_VEL
LIN {X 0,Y 608.442,Z 456.128,A -85,B 0,C 180,E1 -541.986,E2 -541.986} C_VEL
LIN {X 0,Y 608.429,Z 453.745,A -85,B 0,C 180,E1 -542.648,E2 -542.648} C_VEL
LIN {X 0,Y 608.452,Z 448.617,A -85,B 0,C 180,E1 -543.642,E2 -543.642} C_VEL
LIN {X 0,Y 608.452,Z 442.554,A -85,B 0,C 180,E1 -544.472,E2 -544.472} C_VEL
LIN {X 0,Y 608.442,Z 436.249,A -85,B 0,C 180,E1 -545.136,E2 -545.136} C_VEL
LIN {X 0,Y 608.458,Z 429.092,A -85,B 0,C 180,E1 -545.718,E2 -545.718} C_VEL
LIN {X 0,Y 608.443,Z 421.106,A -85,B 0,C 180,E1 -546.217,E2 -546.217} C_VEL
LIN {X 0,Y 608.478,Z 411.444,A -85,B 0,C 180,E1 -546.661,E2 -546.661} C_VEL
LIN {X 0,Y 608.431,Z 403.701,A -85,B 0,C 180,E1 -546.91,E2 -546.91} C_VEL
LIN {X 0,Y 608.412,Z 397.698,A -85,B 0,C 180,E1 -549.134,E2 -549.134} C_VEL
LIN {X 0,Y 607.751,Z 396.282,A -85,B 0,C 180,E1 -549.671,E2 -549.671} C_VEL
LIN {X 0,Y 604.862,Z 394.078,A -85,B 0,C 180,E1 -550.543,E2 -550.543} C_VEL
LIN {X 0,Y 602.428,Z 392.33,A -85,B 0,C 180,E1 -551.245,E2 -551.245} C_VEL
LIN {X 0,Y 601.405,Z 390.951,A -85,B 0,C 180,E1 -551.787,E2 -551.787} C_VEL
LIN {X 0,Y 601.333,Z 390.473,A -85,B 0,C 180,E1 -551.97,E2 -551.97} C_VEL
LIN {X 0,Y 601.361,Z 382.793,A -85,B 0,C 180,E1 -554.899,E2 -554.899} C_VEL
LIN {X 0,Y 601.377,Z 375.574,A -85,B 0,C 180,E1 -557.689,E2 -557.689} C_VEL
LIN {X 0,Y 601.367,Z 368.354,A -85,B 0,C 180,E1 -560.524,E2 -560.524} C_VEL
LIN {X 0,Y 601.38,Z 361.134,A -85,B 0,C 180,E1 -563.412,E2 -563.412} C_VEL
LIN {X 0,Y 601.395,Z 355.127,A -85,B 0,C 180,E1 -565.863,E2 -565.863} C_VEL
LIN {X 0,Y 601.435,Z 348.094,A -85,B 0,C 180,E1 -568.788,E2 -568.788} C_VEL
LIN {X 0,Y 601.423,Z 345.57,A -85,B 0,C 180,E1 -569.865,E2 -569.865} C_VEL
LIN {X 0,Y 601.417,Z 345.571,A -85,B 0,C 180,E1 -572.714,E2 -572.714} C_VEL
LIN {X 0,Y 601.403,Z 345.57,A -85,B 0,C 180,E1 -575.113,E2 -575.113} C_VEL
LIN {X 0,Y 601.437,Z 345.566,A -85,B 0,C 180,E1 -577.419,E2 -577.419} C_VEL
LIN {X 0,Y 601.416,Z 345.569,A -85,B 0,C 180,E1 -579.995,E2 -579.995} C_VEL
LIN {X 0,Y 601.412,Z 345.571,A -85,B 0,C 180,E1 -582.671,E2 -582.671} C_VEL
LIN {X 0,Y 601.431,Z 345.565,A -85,B 0,C 180,E1 -585.482,E2 -585.482} C_VEL
LIN {X 0,Y 601.429,Z 345.567,A -85,B 0,C 180,E1 -588.407,E2 -588.407} C_VEL
LIN {X 0,Y 601.434,Z 345.569,A -85,B 0,C 180,E1 -591.529,E2 -591.529} C_VEL
LIN {X 0,Y 601.388,Z 345.573,A -85,B 0,C 180,E1 -594.245,E2 -594.245} C_VEL
LIN {X 0,Y 601.432,Z 345.567,A -85,B 0,C 180,E1 -596.687,E2 -596.687} C_VEL
LIN {X 0,Y 601.415,Z 345.568,A -85,B 0,C 180,E1 -599.058,E2 -599.058} C_VEL
LIN {X 0,Y 601.439,Z 345.571,A -85,B 0,C 180,E1 -601.373,E2 -601.373} C_VEL
LIN {X 0,Y 601.406,Z 345.569,A -85,B 0,C 180,E1 -603.636,E2 -603.636} C_VEL
LIN {X 0,Y 601.42,Z 345.57,A -85,B 0,C 180,E1 -606.59,E2 -606.59} C_VEL
LIN {X 0,Y 601.437,Z 345.57,A -85,B 0,C 180,E1 -609.478,E2 -609.478} C_VEL
LIN {X 0,Y 601.397,Z 345.57,A -85,B 0,C 180,E1 -612.312,E2 -612.312} C_VEL
LIN {X 0,Y 601.413,Z 345.571,A -85,B 0,C 180,E1 -614.409,E2 -614.409} C_VEL
LIN {X 0,Y 601.417,Z 345.567,A -85,B 0,C 180,E1 -617.172,E2 -617.172} C_VEL
LIN {X 0,Y 601.442,Z 345.568,A -85,B 0,C 180,E1 -619.905,E2 -619.905} C_VEL
LIN {X 0,Y 601.445,Z 345.566,A -85,B 0,C 180,E1 -622.615,E2 -622.615} C_VEL
LIN {X 0,Y 601.42,Z 345.567,A -85,B 0,C 180,E1 -625.308,E2 -625.308} C_VEL
LIN {X 0,Y 601.437,Z 345.572,A -85,B 0,C 180,E1 -627.991,E2 -627.991} C_VEL
LIN {X 0,Y 601.446,Z 345.564,A -85,B 0,C 180,E1 -630.669,E2 -630.669} C_VEL
LIN {X 0,Y 601.429,Z 345.568,A -85,B 0,C 180,E1 -633.35,E2 -633.35} C_VEL
LIN {X 0,Y 601.441,Z 345.567,A -85,B 0,C 180,E1 -636.037,E2 -636.037} C_VEL
LIN {X 0,Y 601.413,Z 345.567,A -85,B 0,C 180,E1 -638.738,E2 -638.738} C_VEL
LIN {X 0,Y 601.427,Z 345.572,A -85,B 0,C 180,E1 -641.458,E2 -641.458} C_VEL
LIN {X 0,Y 601.424,Z 345.568,A -85,B 0,C 180,E1 -644.205,E2 -644.205} C_VEL
LIN {X 0,Y 601.436,Z 345.565,A -85,B 0,C 180,E1 -646.986,E2 -646.986} C_VEL
LIN {X 0,Y 601.403,Z 345.574,A -85,B 0,C 180,E1 -649.81,E2 -649.81} C_VEL
LIN {X 0,Y 601.42,Z 345.568,A -85,B 0,C 180,E1 -652.606,E2 -652.606} C_VEL
LIN {X 0,Y 601.404,Z 345.574,A -85,B 0,C 180,E1 -654.879,E2 -654.879} C_VEL
LIN {X 0,Y 601.423,Z 345.571,A -85,B 0,C 180,E1 -657.867,E2 -657.867} C_VEL
LIN {X 0,Y 601.431,Z 345.567,A -85,B 0,C 180,E1 -660.164,E2 -660.164} C_VEL
LIN {X 0,Y 601.428,Z 345.568,A -85,B 0,C 180,E1 -662.716,E2 -662.716} C_VEL
LIN {X 0,Y 601.403,Z 345.571,A -85,B 0,C 180,E1 -665.112,E2 -665.112} C_VEL
LIN {X 0,Y 601.438,Z 345.565,A -85,B 0,C 180,E1 -667.419,E2 -667.419} C_VEL
LIN {X 0,Y 601.415,Z 345.571,A -85,B 0,C 180,E1 -669.995,E2 -669.995} C_VEL
LIN {X 0,Y 601.416,Z 345.569,A -85,B 0,C 180,E1 -672.67,E2 -672.67} C_VEL
LIN {X 0,Y 601.401,Z 345.569,A -85,B 0,C 180,E1 -675.479,E2 -675.479} C_VEL
LIN {X 0,Y 601.424,Z 345.569,A -85,B 0,C 180,E1 -678.407,E2 -678.407} C_VEL
LIN {X 0,Y 601.435,Z 345.57,A -85,B 0,C 180,E1 -681.529,E2 -681.529} C_VEL
LIN {X 0,Y 601.391,Z 345.571,A -85,B 0,C 180,E1 -684.245,E2 -684.245} C_VEL
LIN {X 0,Y 601.43,Z 345.569,A -85,B 0,C 180,E1 -686.686,E2 -686.686} C_VEL
LIN {X 0,Y 601.419,Z 345.567,A -85,B 0,C 180,E1 -689.058,E2 -689.058} C_VEL
LIN {X 0,Y 601.432,Z 345.572,A -85,B 0,C 180,E1 -691.373,E2 -691.373} C_VEL
LIN {X 0,Y 601.401,Z 345.57,A -85,B 0,C 180,E1 -693.636,E2 -693.636} C_VEL
LIN {X 0,Y 601.422,Z 345.571,A -85,B 0,C 180,E1 -696.59,E2 -696.59} C_VEL
LIN {X 0,Y 601.429,Z 345.569,A -85,B 0,C 180,E1 -699.478,E2 -699.478} C_VEL
LIN {X 0,Y 601.399,Z 345.569,A -85,B 0,C 180,E1 -702.312,E2 -702.312} C_VEL
LIN {X 0,Y 601.413,Z 345.57,A -85,B 0,C 180,E1 -704.409,E2 -704.409} C_VEL
LIN {X 0,Y 601.422,Z 345.566,A -85,B 0,C 180,E1 -707.172,E2 -707.172} C_VEL
LIN {X 0,Y 601.431,Z 345.571,A -85,B 0,C 180,E1 -709.905,E2 -709.905} C_VEL
LIN {X 0,Y 601.445,Z 345.565,A -85,B 0,C 180,E1 -712.615,E2 -712.615} C_VEL
LIN {X 0,Y 601.424,Z 345.567,A -85,B 0,C 180,E1 -715.308,E2 -715.308} C_VEL
LIN {X 0,Y 601.43,Z 345.571,A -85,B 0,C 180,E1 -717.991,E2 -717.991} C_VEL
LIN {X 0,Y 601.45,Z 345.563,A -85,B 0,C 180,E1 -720.669,E2 -720.669} C_VEL
LIN {X 0,Y 601.438,Z 345.568,A -85,B 0,C 180,E1 -723.349,E2 -723.349} C_VEL
LIN {X 0,Y 601.408,Z 345.57,A -85,B 0,C 180,E1 -726.037,E2 -726.037} C_VEL
LIN {X 0,Y 601.416,Z 345.568,A -85,B 0,C 180,E1 -728.738,E2 -728.738} C_VEL
LIN {X 0,Y 601.436,Z 345.572,A -85,B 0,C 180,E1 -731.458,E2 -731.458} C_VEL
LIN {X 0,Y 601.423,Z 345.567,A -85,B 0,C 180,E1 -734.205,E2 -734.205} C_VEL
LIN {X 0,Y 601.434,Z 345.566,A -85,B 0,C 180,E1 -736.986,E2 -736.986} C_VEL
LIN {X 0,Y 601.41,Z 345.576,A -85,B 0,C 180,E1 -739.809,E2 -739.809} C_VEL
LIN {X 0,Y 601.414,Z 345.569,A -85,B 0,C 180,E1 -742.683,E2 -742.683} C_VEL
LIN {X 0,Y 601.406,Z 345.575,A -85,B 0,C 180,E1 -744.878,E2 -744.878} C_VEL
LIN {X 0,Y 601.421,Z 345.566,A -85,B 0,C 180,E1 -747.363,E2 -747.363} C_VEL
LIN {X 0,Y 601.432,Z 345.568,A -85,B 0,C 180,E1 -750.164,E2 -750.164} C_VEL
LIN {X 0,Y 601.419,Z 345.569,A -85,B 0,C 180,E1 -752.715,E2 -752.715} C_VEL
LIN {X 0,Y 601.404,Z 345.572,A -85,B 0,C 180,E1 -755.113,E2 -755.113} C_VEL
LIN {X 0,Y 601.437,Z 345.565,A -85,B 0,C 180,E1 -757.419,E2 -757.419} C_VEL
LIN {X 0,Y 601.405,Z 345.573,A -85,B 0,C 180,E1 -759.996,E2 -759.996} C_VEL
LIN {X 0,Y 601.413,Z 345.569,A -85,B 0,C 180,E1 -762.67,E2 -762.67} C_VEL
LIN {X 0,Y 601.429,Z 345.566,A -85,B 0,C 180,E1 -765.482,E2 -765.482} C_VEL
LIN {X 0,Y 601.428,Z 345.57,A -85,B 0,C 180,E1 -768.407,E2 -768.407} C_VEL
LIN {X 0,Y 601.431,Z 345.573,A -85,B 0,C 180,E1 -771.53,E2 -771.53} C_VEL
LIN {X 0,Y 601.389,Z 345.571,A -85,B 0,C 180,E1 -774.245,E2 -774.245} C_VEL
LIN {X 0,Y 601.431,Z 345.57,A -85,B 0,C 180,E1 -776.687,E2 -776.687} C_VEL
LIN {X 0,Y 601.417,Z 345.567,A -85,B 0,C 180,E1 -779.058,E2 -779.058} C_VEL
LIN {X 0,Y 601.434,Z 345.571,A -85,B 0,C 180,E1 -781.373,E2 -781.373} C_VEL
LIN {X 0,Y 601.433,Z 345.695,A -85,B 0,C 180,E1 -782.201,E2 -782.201} C_VEL
LIN {X 0,Y 601.769,Z 349.898,A -85,B 0,C 180,E1 -782.904,E2 -782.904} C_VEL
LIN {X 0,Y 601.665,Z 367.05,A -85,B 0,C 180,E1 -785.66,E2 -785.66} C_VEL
LIN {X 0,Y 601.598,Z 384.516,A -85,B 0,C 180,E1 -788.408,E2 -788.408} C_VEL
LIN {X 0,Y 601.529,Z 402.275,A -85,B 0,C 180,E1 -791.151,E2 -791.151} C_VEL
LIN {X 0,Y 601.492,Z 421.441,A -85,B 0,C 180,E1 -794.063,E2 -794.063} C_VEL
LIN {X 0,Y 601.437,Z 441.057,A -85,B 0,C 180,E1 -797,E2 -797} C_VEL
LIN {X 0,Y 601.443,Z 448.204,A -85,B 0,C 180,E1 -798.04,E2 -798.04} C_VEL
LIN {X 0,Y 601.583,Z 461.439,A -85,B 0,C 180,E1 -798.267,E2 -798.267} C_VEL
LIN {X 0,Y 601.556,Z 474.222,A -85,B 0,C 180,E1 -798.621,E2 -798.621} C_VEL
LIN {X 0,Y 601.548,Z 485.843,A -85,B 0,C 180,E1 -799.072,E2 -799.072} C_VEL
LIN {X 0,Y 601.483,Z 497.328,A -85,B 0,C 180,E1 -799.651,E2 -799.651} C_VEL
LIN {X 0,Y 601.47,Z 507.931,A -85,B 0,C 180,E1 -800.33,E2 -800.33} C_VEL
LIN {X 0,Y 601.435,Z 517.599,A -85,B 0,C 180,E1 -801.093,E2 -801.093} C_VEL
LIN {X 0,Y 601.406,Z 526.414,A -85,B 0,C 180,E1 -801.939,E2 -801.939} C_VEL
LIN {X 0,Y 601.377,Z 534.999,A -85,B 0,C 180,E1 -802.952,E2 -802.952} C_VEL
LIN {X 0,Y 601.36,Z 541.867,A -85,B 0,C 180,E1 -803.962,E2 -803.962} C_VEL
LIN {X 0,Y 601.345,Z 547.365,A -85,B 0,C 180,E1 -804.971,E2 -804.971} C_VEL
LIN {X 0,Y 601.346,Z 551.676,A -85,B 0,C 180,E1 -805.979,E2 -805.979} C_VEL
LIN {X 0,Y 601.344,Z 553.956,A -85,B 0,C 180,E1 -806.65,E2 -806.65} C_VEL
LIN {X 0,Y 601.325,Z 555.809,A -85,B 0,C 180,E1 -807.32,E2 -807.32} C_VEL
LIN {X 0,Y 601.343,Z 557.202,A -85,B 0,C 180,E1 -807.991,E2 -807.991} C_VEL
LIN {X 0,Y 601.339,Z 558.784,A -85,B 0,C 180,E1 -809.33,E2 -809.33} C_VEL
LIN {X 0,Y 601.335,Z 559,A -85,B 0,C 180,E1 -810,E2 -810} C_VEL
LIN {X 0,Y 601.348,Z 558.184,A -85,B 0,C 180,E1 -811.339,E2 -811.339} C_VEL
LIN {X 0,Y 601.343,Z 557.202,A -85,B 0,C 180,E1 -812.009,E2 -812.009} C_VEL
LIN {X 0,Y 601.325,Z 555.809,A -85,B 0,C 180,E1 -812.68,E2 -812.68} C_VEL
LIN {X 0,Y 601.367,Z 552.896,A -85,B 0,C 180,E1 -813.685,E2 -813.685} C_VEL
LIN {X 0,Y 601.336,Z 548.95,A -85,B 0,C 180,E1 -814.693,E2 -814.693} C_VEL
LIN {X 0,Y 601.372,Z 542.876,A -85,B 0,C 180,E1 -815.869,E2 -815.869} C_VEL
LIN {X 0,Y 601.382,Z 536.235,A -85,B 0,C 180,E1 -816.88,E2 -816.88} C_VEL
LIN {X 0,Y 601.4,Z 527.989,A -85,B 0,C 180,E1 -817.892,E2 -817.892} C_VEL
LIN {X 0,Y 601.436,Z 519.536,A -85,B 0,C 180,E1 -818.738,E2 -818.738} C_VEL
LIN {X 0,Y 601.451,Z 509.091,A -85,B 0,C 180,E1 -819.585,E2 -819.585} C_VEL
LIN {X 0,Y 601.471,Z 498.755,A -85,B 0,C 180,E1 -820.265,E2 -820.265} C_VEL
LIN {X 0,Y 601.539,Z 486.58,A -85,B 0,C 180,E1 -820.897,E2 -820.897} C_VEL
LIN {X 0,Y 601.556,Z 474.212,A -85,B 0,C 180,E1 -821.379,E2 -821.379} C_VEL
LIN {X 0,Y 601.583,Z 461.433,A -85,B 0,C 180,E1 -821.733,E2 -821.733} C_VEL
LIN {X 0,Y 601.424,Z 447.98,A -85,B 0,C 180,E1 -821.971,E2 -821.971} C_VEL
LIN {X 0,Y 601.478,Z 428.364,A -85,B 0,C 180,E1 -824.896,E2 -824.896} C_VEL
LIN {X 0,Y 601.511,Z 411.055,A -85,B 0,C 180,E1 -827.509,E2 -827.509} C_VEL
LIN {X 0,Y 601.583,Z 393.746,A -85,B 0,C 180,E1 -830.16,E2 -830.16} C_VEL
LIN {X 0,Y 601.635,Z 375.284,A -85,B 0,C 180,E1 -833.037,E2 -833.037} C_VEL
LIN {X 0,Y 601.733,Z 357.106,A -85,B 0,C 180,E1 -835.93,E2 -835.93} C_VEL
LIN {X 0,Y 601.706,Z 346.93,A -85,B 0,C 180,E1 -837.583,E2 -837.583} C_VEL
LIN {X 0,Y 601.427,Z 345.574,A -85,B 0,C 180,E1 -837.833,E2 -837.833} C_VEL
LIN {X 0,Y 601.432,Z 345.571,A -85,B 0,C 180,E1 -840.164,E2 -840.164} C_VEL
LIN {X 0,Y 601.43,Z 345.57,A -85,B 0,C 180,E1 -842.716,E2 -842.716} C_VEL
LIN {X 0,Y 601.398,Z 345.576,A -85,B 0,C 180,E1 -845.112,E2 -845.112} C_VEL
LIN {X 0,Y 601.437,Z 345.572,A -85,B 0,C 180,E1 -847.419,E2 -847.419} C_VEL
LIN {X 0,Y 601.404,Z 345.573,A -85,B 0,C 180,E1 -849.996,E2 -849.996} C_VEL
LIN {X 0,Y 601.416,Z 345.574,A -85,B 0,C 180,E1 -852.67,E2 -852.67} C_VEL
LIN {X 0,Y 601.43,Z 345.571,A -85,B 0,C 180,E1 -855.482,E2 -855.482} C_VEL
LIN {X 0,Y 601.429,Z 345.57,A -85,B 0,C 180,E1 -858.407,E2 -858.407} C_VEL
LIN {X 0,Y 601.44,Z 345.57,A -85,B 0,C 180,E1 -860.876,E2 -860.876} C_VEL
LIN {X 0,Y 601.411,Z 345.573,A -85,B 0,C 180,E1 -863.739,E2 -863.739} C_VEL
LIN {X 0,Y 601.43,Z 345.57,A -85,B 0,C 180,E1 -866.687,E2 -866.687} C_VEL
LIN {X 0,Y 601.418,Z 345.572,A -85,B 0,C 180,E1 -869.058,E2 -869.058} C_VEL
LIN {X 0,Y 601.431,Z 345.657,A -85,B 0,C 180,E1 -870.319,E2 -870.319} C_VEL
LIN {X 0,Y 601.421,Z 351.942,A -85,B 0,C 180,E1 -872.887,E2 -872.887} C_VEL
LIN {X 0,Y 601.405,Z 358.758,A -85,B 0,C 180,E1 -875.715,E2 -875.715} C_VEL
LIN {X 0,Y 601.362,Z 364.52,A -85,B 0,C 180,E1 -878.039,E2 -878.039} C_VEL
LIN {X 0,Y 601.375,Z 371.735,A -85,B 0,C 180,E1 -880.9,E2 -880.9} C_VEL
LIN {X 0,Y 601.358,Z 378.951,A -85,B 0,C 180,E1 -883.711,E2 -883.711} C_VEL
LIN {X 0,Y 601.344,Z 386.167,A -85,B 0,C 180,E1 -886.482,E2 -886.482} C_VEL
LIN {X 0,Y 601.346,Z 393.384,A -85,B 0,C 180,E1 -889.223,E2 -889.223} C_VEL
LIN {X 0,Y 601.325,Z 400.601,A -85,B 0,C 180,E1 -891.938,E2 -891.938} C_VEL
LIN {X 0,Y 601.343,Z 403.681,A -85,B 0,C 180,E1 -893.091,E2 -893.091} C_VEL
LIN {X 0,Y 601.433,Z 413.835,A -85,B 0,C 180,E1 -893.446,E2 -893.446} C_VEL
LIN {X 0,Y 601.387,Z 422.181,A -85,B 0,C 180,E1 -893.861,E2 -893.861} C_VEL
LIN {X 0,Y 601.381,Z 430.191,A -85,B 0,C 180,E1 -894.383,E2 -894.383} C_VEL
LIN {X 0,Y 601.364,Z 437.033,A -85,B 0,C 180,E1 -894.972,E2 -894.972} C_VEL
LIN {X 0,Y 601.362,Z 443.211,A -85,B 0,C 180,E1 -895.643,E2 -895.643} C_VEL
LIN {X 0,Y 601.374,Z 448.071,A -85,B 0,C 180,E1 -896.315,E2 -896.315} C_VEL
LIN {X 0,Y 601.379,Z 451.821,A -85,B 0,C 180,E1 -896.986,E2 -896.986} C_VEL
LIN {X 0,Y 601.343,Z 455.827,A -85,B 0,C 180,E1 -897.991,E2 -897.991} C_VEL
LIN {X 0,Y 601.347,Z 457.57,A -85,B 0,C 180,E1 -898.661,E2 -898.661} C_VEL
LIN {X 0,Y 601.341,Z 458.616,A -85,B 0,C 180,E1 -899.33,E2 -899.33} C_VEL
LIN {X 0,Y 601.335,Z 458.996,A -85,B 0,C 180,E1 -900,E2 -900} C_VEL
LIN {X 0,Y 601.339,Z 458.714,A -85,B 0,C 180,E1 -900.67,E2 -900.67} C_VEL
LIN {X 0,Y 601.349,Z 457.767,A -85,B 0,C 180,E1 -901.339,E2 -901.339} C_VEL
LIN {X 0,Y 601.342,Z 456.127,A -85,B 0,C 180,E1 -902.009,E2 -902.009} C_VEL
LIN {X 0,Y 601.332,Z 453.742,A -85,B 0,C 180,E1 -902.68,E2 -902.68} C_VEL
LIN {X 0,Y 601.375,Z 448.615,A -85,B 0,C 180,E1 -903.685,E2 -903.685} C_VEL
LIN {X 0,Y 601.378,Z 442.55,A -85,B 0,C 180,E1 -904.524,E2 -904.524} C_VEL
LIN {X 0,Y 601.36,Z 436.243,A -85,B 0,C 180,E1 -905.197,E2 -905.197} C_VEL
LIN {X 0,Y 601.391,Z 429.086,A -85,B 0,C 180,E1 -905.785,E2 -905.785} C_VEL
LIN {X 0,Y 601.402,Z 420.636,A -85,B 0,C 180,E1 -906.316,E2 -906.316} C_VEL
LIN {X 0,Y 601.427,Z 411.074,A -85,B 0,C 180,E1 -906.753,E2 -906.753} C_VEL
LIN {X 0,Y 601.337,Z 403.66,A -85,B 0,C 180,E1 -907.007,E2 -907.007} C_VEL
LIN {X 0,Y 601.332,Z 397.231,A -85,B 0,C 180,E1 -909.417,E2 -909.417} C_VEL
LIN {X 0,Y 601.333,Z 390.473,A -85,B 0,C 180,E1 -911.97,E2 -911.97} C_VEL
LIN {X 0,Y 600.695,Z 389.077,A -85,B 0,C 180,E1 -912.513,E2 -912.513} C_VEL
LIN {X 0,Y 597.834,Z 386.928,A -85,B 0,C 180,E1 -913.397,E2 -913.397} C_VEL
LIN {X 0,Y 595.4,Z 385.228,A -85,B 0,C 180,E1 -914.108,E2 -914.108} C_VEL
LIN {X 0,Y 594.357,Z 383.878,A -85,B 0,C 180,E1 -914.657,E2 -914.657} C_VEL
LIN {X 0,Y 594.273,Z 383.406,A -85,B 0,C 180,E1 -914.842,E2 -914.842} C_VEL
LIN {X 0,Y 594.298,Z 377.377,A -85,B 0,C 180,E1 -917.196,E2 -917.196} C_VEL
LIN {X 0,Y 594.293,Z 370.158,A -85,B 0,C 180,E1 -920.057,E2 -920.057} C_VEL
LIN {X 0,Y 594.302,Z 362.938,A -85,B 0,C 180,E1 -922.97,E2 -922.97} C_VEL
LIN {X 0,Y 594.337,Z 357.522,A -85,B 0,C 180,E1 -925.195,E2 -925.195} C_VEL
LIN {X 0,Y 594.353,Z 352.07,A -85,B 0,C 180,E1 -927.52,E2 -927.52} C_VEL
LIN {X 0,Y 594.394,Z 346.445,A -85,B 0,C 180,E1 -929.863,E2 -929.863} C_VEL
LIN {X 0,Y 594.366,Z 346.445,A -85,B 0,C 180,E1 -932.147,E2 -932.147} C_VEL
LIN {X 0,Y 594.389,Z 346.45,A -85,B 0,C 180,E1 -934.58,E2 -934.58} C_VEL
LIN {X 0,Y 594.389,Z 346.443,A -85,B 0,C 180,E1 -937.087,E2 -937.087} C_VEL
LIN {X 0,Y 594.381,Z 346.449,A -85,B 0,C 180,E1 -939.774,E2 -939.774} C_VEL
LIN {X 0,Y 594.369,Z 346.446,A -85,B 0,C 180,E1 -942.376,E2 -942.376} C_VEL
LIN {X 0,Y 594.36,Z 346.447,A -85,B 0,C 180,E1 -945.192,E2 -945.192} C_VEL
LIN {X 0,Y 594.375,Z 346.447,A -85,B 0,C 180,E1 -947.625,E2 -947.625} C_VEL
LIN {X 0,Y 594.374,Z 346.445,A -85,B 0,C 180,E1 -950.319,E2 -950.319} C_VEL
LIN {X 0,Y 594.388,Z 346.45,A -85,B 0,C 180,E1 -952.913,E2 -952.913} C_VEL
LIN {X 0,Y 594.384,Z 346.445,A -85,B 0,C 180,E1 -955.862,E2 -955.862} C_VEL
LIN {X 0,Y 594.374,Z 346.445,A -85,B 0,C 180,E1 -958.65,E2 -958.65} C_VEL
LIN {X 0,Y 594.389,Z 346.446,A -85,B 0,C 180,E1 -961.042,E2 -961.042} C_VEL
LIN {X 0,Y 594.39,Z 346.443,A -85,B 0,C 180,E1 -963.977,E2 -963.977} C_VEL
LIN {X 0,Y 594.389,Z 346.45,A -85,B 0,C 180,E1 -966.296,E2 -966.296} C_VEL
LIN {X 0,Y 594.41,Z 346.442,A -85,B 0,C 180,E1 -969.225,E2 -969.225} C_VEL
LIN {X 0,Y 594.355,Z 346.447,A -85,B 0,C 180,E1 -972.095,E2 -972.095} C_VEL
LIN {X 0,Y 594.367,Z 346.447,A -85,B 0,C 180,E1 -974.219,E2 -974.219} C_VEL
LIN {X 0,Y 594.383,Z 346.451,A -85,B 0,C 180,E1 -976.321,E2 -976.321} C_VEL
LIN {X 0,Y 594.38,Z 346.444,A -85,B 0,C 180,E1 -979.095,E2 -979.095} C_VEL
LIN {X 0,Y 594.418,Z 346.44,A -85,B 0,C 180,E1 -981.843,E2 -981.843} C_VEL
LIN {X 0,Y 594.404,Z 346.447,A -85,B 0,C 180,E1 -984.572,E2 -984.572} C_VEL
LIN {X 0,Y 594.405,Z 346.441,A -85,B 0,C 180,E1 -987.289,E2 -987.289} C_VEL
LIN {X 0,Y 594.419,Z 346.442,A -85,B 0,C 180,E1 -990,E2 -990} C_VEL
LIN {X 0,Y 594.405,Z 346.444,A -85,B 0,C 180,E1 -992.711,E2 -992.711} C_VEL
LIN {X 0,Y 594.396,Z 346.442,A -85,B 0,C 180,E1 -995.428,E2 -995.428} C_VEL
LIN {X 0,Y 594.417,Z 346.444,A -85,B 0,C 180,E1 -998.157,E2 -998.157} C_VEL
LIN {X 0,Y 594.393,Z 346.445,A -85,B 0,C 180,E1 -1001.073,E2 -1001.073} C_VEL
LIN {X 0,Y 594.386,Z 346.443,A -85,B 0,C 180,E1 -1003.679,E2 -1003.679} C_VEL
LIN {X 0,Y 594.402,Z 346.443,A -85,B 0,C 180,E1 -1006.72,E2 -1006.72} C_VEL
LIN {X 0,Y 594.368,Z 346.447,A -85,B 0,C 180,E1 -1009.334,E2 -1009.334} C_VEL
LIN {X 0,Y 594.37,Z 346.45,A -85,B 0,C 180,E1 -1011.503,E2 -1011.503} C_VEL
LIN {X 0,Y 594.393,Z 346.446,A -85,B 0,C 180,E1 -1014.446,E2 -1014.446} C_VEL
LIN {X 0,Y 594.385,Z 346.446,A -85,B 0,C 180,E1 -1016.7,E2 -1016.7} C_VEL
LIN {X 0,Y 594.385,Z 346.443,A -85,B 0,C 180,E1 -1018.998,E2 -1018.998} C_VEL
LIN {X 0,Y 594.38,Z 346.447,A -85,B 0,C 180,E1 -1021.642,E2 -1021.642} C_VEL
LIN {X 0,Y 594.387,Z 346.448,A -85,B 0,C 180,E1 -1024.58,E2 -1024.58} C_VEL
LIN {X 0,Y 594.393,Z 346.444,A -85,B 0,C 180,E1 -1027.608,E2 -1027.608} C_VEL
LIN {X 0,Y 594.369,Z 346.445,A -85,B 0,C 180,E1 -1030.567,E2 -1030.567} C_VEL
LIN {X 0,Y 594.371,Z 346.449,A -85,B 0,C 180,E1 -1033.299,E2 -1033.299} C_VEL
LIN {X 0,Y 594.363,Z 346.45,A -85,B 0,C 180,E1 -1036.161,E2 -1036.161} C_VEL
LIN {X 0,Y 594.381,Z 346.445,A -85,B 0,C 180,E1 -1038.536,E2 -1038.536} C_VEL
LIN {X 0,Y 594.386,Z 346.449,A -85,B 0,C 180,E1 -1041.296,E2 -1041.296} C_VEL
LIN {X 0,Y 594.355,Z 346.447,A -85,B 0,C 180,E1 -1043.755,E2 -1043.755} C_VEL
LIN {X 0,Y 594.384,Z 346.448,A -85,B 0,C 180,E1 -1046.239,E2 -1046.239} C_VEL
LIN {X 0,Y 594.373,Z 346.445,A -85,B 0,C 180,E1 -1048.65,E2 -1048.65} C_VEL
LIN {X 0,Y 594.386,Z 346.445,A -85,B 0,C 180,E1 -1051.042,E2 -1051.042} C_VEL
LIN {X 0,Y 594.387,Z 346.447,A -85,B 0,C 180,E1 -1053.3,E2 -1053.3} C_VEL
LIN {X 0,Y 594.393,Z 346.448,A -85,B 0,C 180,E1 -1056.296,E2 -1056.296} C_VEL
LIN {X 0,Y 594.402,Z 346.442,A -85,B 0,C 180,E1 -1059.224,E2 -1059.224} C_VEL
LIN {X 0,Y 594.356,Z 346.447,A -85,B 0,C 180,E1 -1062.095,E2 -1062.095} C_VEL
LIN {X 0,Y 594.366,Z 346.446,A -85,B 0,C 180,E1 -1064.219,E2 -1064.219} C_VEL
LIN {X 0,Y 594.383,Z 346.449,A -85,B 0,C 180,E1 -1066.321,E2 -1066.321} C_VEL
LIN {X 0,Y 594.376,Z 346.445,A -85,B 0,C 180,E1 -1069.095,E2 -1069.095} C_VEL
LIN {X 0,Y 594.417,Z 346.441,A -85,B 0,C 180,E1 -1071.843,E2 -1071.843} C_VEL
LIN {X 0,Y 594.398,Z 346.446,A -85,B 0,C 180,E1 -1074.572,E2 -1074.572} C_VEL
LIN {X 0,Y 594.41,Z 346.44,A -85,B 0,C 180,E1 -1077.289,E2 -1077.289} C_VEL
LIN {X 0,Y 594.418,Z 346.443,A -85,B 0,C 180,E1 -1080,E2 -1080} C_VEL
LIN {X 0,Y 594.415,Z 346.441,A -85,B 0,C 180,E1 -1082.711,E2 -1082.711} C_VEL
LIN {X 0,Y 594.392,Z 346.442,A -85,B 0,C 180,E1 -1085.428,E2 -1085.428} C_VEL
LIN {X 0,Y 594.395,Z 346.442,A -85,B 0,C 180,E1 -1087.473,E2 -1087.473} C_VEL
LIN {X 0,Y 594.398,Z 346.443,A -85,B 0,C 180,E1 -1090.216,E2 -1090.216} C_VEL
LIN {X 0,Y 594.372,Z 346.45,A -85,B 0,C 180,E1 -1092.983,E2 -1092.983} C_VEL
LIN {X 0,Y 594.376,Z 346.448,A -85,B 0,C 180,E1 -1095.078,E2 -1095.078} C_VEL
LIN {X 0,Y 594.392,Z 346.442,A -85,B 0,C 180,E1 -1097.193,E2 -1097.193} C_VEL
LIN {X 0,Y 594.377,Z 346.448,A -85,B 0,C 180,E1 -1100.054,E2 -1100.054} C_VEL
LIN {X 0,Y 594.359,Z 346.451,A -85,B 0,C 180,E1 -1102.968,E2 -1102.968} C_VEL
LIN {X 0,Y 594.376,Z 346.446,A -85,B 0,C 180,E1 -1105.193,E2 -1105.193} C_VEL
LIN {X 0,Y 594.389,Z 346.443,A -85,B 0,C 180,E1 -1107.527,E2 -1107.527} C_VEL
LIN {X 0,Y 594.39,Z 346.443,A -85,B 0,C 180,E1 -1110.328,E2 -1110.328} C_VEL
LIN {X 0,Y 594.38,Z 346.448,A -85,B 0,C 180,E1 -1112.95,E2 -1112.95} C_VEL
LIN {X 0,Y 594.36,Z 346.447,A -85,B 0,C 180,E1 -1115.408,E2 -1115.408} C_VEL
LIN {X 0,Y 594.393,Z 346.446,A -85,B 0,C 180,E1 -1117.94,E2 -1117.94} C_VEL
LIN {X 0,Y 594.377,Z 346.444,A -85,B 0,C 180,E1 -1120.822,E2 -1120.822} C_VEL
LIN {X 0,Y 594.385,Z 346.443,A -85,B 0,C 180,E1 -1123.841,E2 -1123.841} C_VEL
LIN {X 0,Y 594.383,Z 346.448,A -85,B 0,C 180,E1 -1126.702,E2 -1126.702} C_VEL
LIN {X 0,Y 594.372,Z 346.447,A -85,B 0,C 180,E1 -1129.433,E2 -1129.433} C_VEL
LIN {X 0,Y 594.391,Z 346.442,A -85,B 0,C 180,E1 -1132.392,E2 -1132.392} C_VEL
LIN {X 0,Y 594.384,Z 346.444,A -85,B 0,C 180,E1 -1135.42,E2 -1135.42} C_VEL
LIN {X 0,Y 594.382,Z 346.448,A -85,B 0,C 180,E1 -1138.357,E2 -1138.357} C_VEL
LIN {X 0,Y 594.386,Z 346.446,A -85,B 0,C 180,E1 -1141.042,E2 -1141.042} C_VEL
LIN {X 0,Y 594.425,Z 346.601,A -85,B 0,C 180,E1 -1141.995,E2 -1141.995} C_VEL
LIN {X 0,Y 594.889,Z 349.898,A -85,B 0,C 180,E1 -1142.565,E2 -1142.565} C_VEL
LIN {X 0,Y 594.786,Z 366.284,A -85,B 0,C 180,E1 -1145.236,E2 -1145.236} C_VEL
LIN {X 0,Y 594.659,Z 384.516,A -85,B 0,C 180,E1 -1148.143,E2 -1148.143} C_VEL
LIN {X 0,Y 594.581,Z 402.158,A -85,B 0,C 180,E1 -1150.904,E2 -1150.904} C_VEL
LIN {X 0,Y 594.489,Z 421.441,A -85,B 0,C 180,E1 -1153.87,E2 -1153.87} C_VEL
LIN {X 0,Y 594.422,Z 439.904,A -85,B 0,C 180,E1 -1156.67,E2 -1156.67} C_VEL
LIN {X 0,Y 594.401,Z 448.204,A -85,B 0,C 180,E1 -1157.896,E2 -1157.896} C_VEL
LIN {X 0,Y 594.646,Z 454.947,A -85,B 0,C 180,E1 -1157.999,E2 -1157.999} C_VEL
LIN {X 0,Y 594.603,Z 468.217,A -85,B 0,C 180,E1 -1158.3,E2 -1158.3} C_VEL
LIN {X 0,Y 594.599,Z 480.417,A -85,B 0,C 180,E1 -1158.713,E2 -1158.713} C_VEL
LIN {X 0,Y 594.529,Z 492.633,A -85,B 0,C 180,E1 -1159.27,E2 -1159.27} C_VEL
LIN {X 0,Y 594.48,Z 504.199,A -85,B 0,C 180,E1 -1159.958,E2 -1159.958} C_VEL
LIN {X 0,Y 594.414,Z 514.596,A -85,B 0,C 180,E1 -1160.73,E2 -1160.73} C_VEL
LIN {X 0,Y 594.383,Z 523.112,A -85,B 0,C 180,E1 -1161.501,E2 -1161.501} C_VEL
LIN {X 0,Y 594.347,Z 530.96,A -85,B 0,C 180,E1 -1162.355,E2 -1162.355} C_VEL
LIN {X 0,Y 594.282,Z 538.813,A -85,B 0,C 180,E1 -1163.408,E2 -1163.408} C_VEL
LIN {X 0,Y 594.289,Z 545.681,A -85,B 0,C 180,E1 -1164.571,E2 -1164.571} C_VEL
LIN {X 0,Y 594.27,Z 550.371,A -85,B 0,C 180,E1 -1165.591,E2 -1165.591} C_VEL
LIN {X 0,Y 594.267,Z 553.956,A -85,B 0,C 180,E1 -1166.61,E2 -1166.61} C_VEL
LIN {X 0,Y 594.226,Z 555.809,A -85,B 0,C 180,E1 -1167.288,E2 -1167.288} C_VEL
LIN {X 0,Y 594.242,Z 557.201,A -85,B 0,C 180,E1 -1167.967,E2 -1167.967} C_VEL
LIN {X 0,Y 594.239,Z 558.784,A -85,B 0,C 180,E1 -1169.322,E2 -1169.322} C_VEL
LIN {X 0,Y 594.236,Z 559,A -85,B 0,C 180,E1 -1170,E2 -1170} C_VEL
LIN {X 0,Y 594.248,Z 558.185,A -85,B 0,C 180,E1 -1171.355,E2 -1171.355} C_VEL
LIN {X 0,Y 594.242,Z 557.202,A -85,B 0,C 180,E1 -1172.033,E2 -1172.033} C_VEL
LIN {X 0,Y 594.226,Z 555.809,A -85,B 0,C 180,E1 -1172.712,E2 -1172.712} C_VEL
LIN {X 0,Y 594.288,Z 552.896,A -85,B 0,C 180,E1 -1173.729,E2 -1173.729} C_VEL
LIN {X 0,Y 594.241,Z 548.949,A -85,B 0,C 180,E1 -1174.749,E2 -1174.749} C_VEL
LIN {X 0,Y 594.304,Z 542.877,A -85,B 0,C 180,E1 -1175.939,E2 -1175.939} C_VEL
LIN {X 0,Y 594.308,Z 536.235,A -85,B 0,C 180,E1 -1176.962,E2 -1176.962} C_VEL
LIN {X 0,Y 594.359,Z 527.989,A -85,B 0,C 180,E1 -1177.986,E2 -1177.986} C_VEL
LIN {X 0,Y 594.382,Z 519.536,A -85,B 0,C 180,E1 -1178.842,E2 -1178.842} C_VEL
LIN {X 0,Y 594.435,Z 509.092,A -85,B 0,C 180,E1 -1179.699,E2 -1179.699} C_VEL
LIN {X 0,Y 594.484,Z 498.757,A -85,B 0,C 180,E1 -1180.386,E2 -1180.386} C_VEL
LIN {X 0,Y 594.559,Z 487.705,A -85,B 0,C 180,E1 -1180.974,E2 -1180.974} C_VEL
LIN {X 0,Y 594.58,Z 475.703,A -85,B 0,C 180,E1 -1181.464,E2 -1181.464} C_VEL
LIN {X 0,Y 594.636,Z 462.347,A -85,B 0,C 180,E1 -1181.85,E2 -1181.85} C_VEL
LIN {X 0,Y 594.511,Z 449.076,A -85,B 0,C 180,E1 -1182.091,E2 -1182.091} C_VEL
LIN {X 0,Y 594.384,Z 447.98,A -85,B 0,C 180,E1 -1182.115,E2 -1182.115} C_VEL
LIN {X 0,Y 594.46,Z 428.364,A -85,B 0,C 180,E1 -1185.076,E2 -1185.076} C_VEL
LIN {X 0,Y 594.528,Z 411.055,A -85,B 0,C 180,E1 -1187.722,E2 -1187.722} C_VEL
LIN {X 0,Y 594.617,Z 393.746,A -85,B 0,C 180,E1 -1190.406,E2 -1190.406} C_VEL
LIN {X 0,Y 594.704,Z 375.284,A -85,B 0,C 180,E1 -1193.322,E2 -1193.322} C_VEL
LIN {X 0,Y 594.848,Z 357.959,A -85,B 0,C 180,E1 -1196.113,E2 -1196.113} C_VEL
LIN {X 0,Y 594.875,Z 348.807,A -85,B 0,C 180,E1 -1197.616,E2 -1197.616} C_VEL
LIN {X 0,Y 594.402,Z 346.448,A -85,B 0,C 180,E1 -1198.051,E2 -1198.051} C_VEL
LIN {X 0,Y 594.385,Z 346.448,A -85,B 0,C 180,E1 -1200.56,E2 -1200.56} C_VEL
LIN {X 0,Y 594.384,Z 346.449,A -85,B 0,C 180,E1 -1202.95,E2 -1202.95} C_VEL
LIN {X 0,Y 594.353,Z 346.453,A -85,B 0,C 180,E1 -1205.409,E2 -1205.409} C_VEL
LIN {X 0,Y 594.384,Z 346.448,A -85,B 0,C 180,E1 -1207.941,E2 -1207.941} C_VEL
LIN {X 0,Y 594.38,Z 346.449,A -85,B 0,C 180,E1 -1210.822,E2 -1210.822} C_VEL
LIN {X 0,Y 594.386,Z 346.449,A -85,B 0,C 180,E1 -1213.841,E2 -1213.841} C_VEL
LIN {X 0,Y 594.384,Z 346.45,A -85,B 0,C 180,E1 -1216.702,E2 -1216.702} C_VEL
LIN {X 0,Y 594.373,Z 346.449,A -85,B 0,C 180,E1 -1219.433,E2 -1219.433} C_VEL
LIN {X 0,Y 594.392,Z 346.447,A -85,B 0,C 180,E1 -1222.392,E2 -1222.392} C_VEL
LIN {X 0,Y 594.389,Z 346.449,A -85,B 0,C 180,E1 -1225.421,E2 -1225.421} C_VEL
LIN {X 0,Y 594.382,Z 346.451,A -85,B 0,C 180,E1 -1228.357,E2 -1228.357} C_VEL
LIN {X 0,Y 594.411,Z 346.56,A -85,B 0,C 180,E1 -1230.323,E2 -1230.323} C_VEL
LIN {X 0,Y 594.373,Z 353.899,A -85,B 0,C 180,E1 -1233.3,E2 -1233.3} C_VEL
LIN {X 0,Y 594.34,Z 359.172,A -85,B 0,C 180,E1 -1235.577,E2 -1235.577} C_VEL
LIN {X 0,Y 594.319,Z 364.521,A -85,B 0,C 180,E1 -1237.765,E2 -1237.765} C_VEL
LIN {X 0,Y 594.293,Z 371.737,A -85,B 0,C 180,E1 -1240.663,E2 -1240.663} C_VEL
LIN {X 0,Y 594.304,Z 378.953,A -85,B 0,C 180,E1 -1243.512,E2 -1243.512} C_VEL
LIN {X 0,Y 594.26,Z 386.169,A -85,B 0,C 180,E1 -1246.318,E2 -1246.318} C_VEL
LIN {X 0,Y 594.243,Z 393.385,A -85,B 0,C 180,E1 -1249.092,E2 -1249.092} C_VEL
LIN {X 0,Y 594.252,Z 400.602,A -85,B 0,C 180,E1 -1251.841,E2 -1251.841} C_VEL
LIN {X 0,Y 594.249,Z 403.703,A -85,B 0,C 180,E1 -1253.016,E2 -1253.016} C_VEL
LIN {X 0,Y 594.397,Z 412.602,A -85,B 0,C 180,E1 -1253.314,E2 -1253.314} C_VEL
LIN {X 0,Y 594.354,Z 420.807,A -85,B 0,C 180,E1 -1253.709,E2 -1253.709} C_VEL
LIN {X 0,Y 594.32,Z 429.012,A -85,B 0,C 180,E1 -1254.231,E2 -1254.231} C_VEL
LIN {X 0,Y 594.289,Z 437.039,A -85,B 0,C 180,E1 -1254.912,E2 -1254.912} C_VEL
LIN {X 0,Y 594.286,Z 443.215,A -85,B 0,C 180,E1 -1255.591,E2 -1255.591} C_VEL
LIN {X 0,Y 594.299,Z 448.074,A -85,B 0,C 180,E1 -1256.271,E2 -1256.271} C_VEL
LIN {X 0,Y 594.278,Z 451.823,A -85,B 0,C 180,E1 -1256.949,E2 -1256.949} C_VEL
LIN {X 0,Y 594.244,Z 455.83,A -85,B 0,C 180,E1 -1257.967,E2 -1257.967} C_VEL
LIN {X 0,Y 594.247,Z 457.572,A -85,B 0,C 180,E1 -1258.645,E2 -1258.645} C_VEL
LIN {X 0,Y 594.241,Z 458.617,A -85,B 0,C 180,E1 -1259.322,E2 -1259.322} C_VEL
LIN {X 0,Y 594.236,Z 458.996,A -85,B 0,C 180,E1 -1260,E2 -1260} C_VEL
LIN {X 0,Y 594.239,Z 458.713,A -85,B 0,C 180,E1 -1260.678,E2 -1260.678} C_VEL
LIN {X 0,Y 594.249,Z 457.766,A -85,B 0,C 180,E1 -1261.355,E2 -1261.355} C_VEL
LIN {X 0,Y 594.242,Z 456.125,A -85,B 0,C 180,E1 -1262.033,E2 -1262.033} C_VEL
LIN {X 0,Y 594.237,Z 453.74,A -85,B 0,C 180,E1 -1262.712,E2 -1262.712} C_VEL
LIN {X 0,Y 594.3,Z 448.612,A -85,B 0,C 180,E1 -1263.729,E2 -1263.729} C_VEL
LIN {X 0,Y 594.31,Z 442.546,A -85,B 0,C 180,E1 -1264.578,E2 -1264.578} C_VEL
LIN {X 0,Y 594.279,Z 436.237,A -85,B 0,C 180,E1 -1265.259,E2 -1265.259} C_VEL
LIN {X 0,Y 594.315,Z 429.08,A -85,B 0,C 180,E1 -1265.854,E2 -1265.854} C_VEL
LIN {X 0,Y 594.351,Z 420.354,A -85,B 0,C 180,E1 -1266.407,E2 -1266.407} C_VEL
LIN {X 0,Y 594.4,Z 411.06,A -85,B 0,C 180,E1 -1266.833,E2 -1266.833} C_VEL
LIN {X 0,Y 594.247,Z 403.659,A -85,B 0,C 180,E1 -1267.091,E2 -1267.091} C_VEL
LIN {X 0,Y 594.251,Z 397.23,A -85,B 0,C 180,E1 -1269.531,E2 -1269.531} C_VEL
LIN {X 0,Y 594.247,Z 390.011,A -85,B 0,C 180,E1 -1272.291,E2 -1272.291} C_VEL
LIN {X 0,Y 594.273,Z 383.406,A -85,B 0,C 180,E1 -1274.842,E2 -1274.842} C_VEL
LIN {X 0,Y 593.611,Z 382.036,A -85,B 0,C 180,E1 -1275.392,E2 -1275.392} C_VEL
LIN {X 0,Y 590.751,Z 379.946,A -85,B 0,C 180,E1 -1276.289,E2 -1276.289} C_VEL
LIN {X 0,Y 588.33,Z 378.296,A -85,B 0,C 180,E1 -1277.011,E2 -1277.011} C_VEL
LIN {X 0,Y 587.286,Z 376.978,A -85,B 0,C 180,E1 -1277.567,E2 -1277.567} C_VEL
LIN {X 0,Y 587.198,Z 376.514,A -85,B 0,C 180,E1 -1277.754,E2 -1277.754} C_VEL
LIN {X 0,Y 587.214,Z 370.156,A -85,B 0,C 180,E1 -1280.309,E2 -1280.309} C_VEL
LIN {X 0,Y 587.247,Z 363.932,A -85,B 0,C 180,E1 -1282.851,E2 -1282.851} C_VEL
LIN {X 0,Y 587.301,Z 357.669,A -85,B 0,C 180,E1 -1285.518,E2 -1285.518} C_VEL
LIN {X 0,Y 587.301,Z 352.21,A -85,B 0,C 180,E1 -1287.82,E2 -1287.82} C_VEL
LIN {X 0,Y 587.363,Z 347.321,A -85,B 0,C 180,E1 -1289.872,E2 -1289.872} C_VEL
LIN {X 0,Y 587.339,Z 347.323,A -85,B 0,C 180,E1 -1292.579,E2 -1292.579} C_VEL
LIN {X 0,Y 587.334,Z 347.323,A -85,B 0,C 180,E1 -1295.055,E2 -1295.055} C_VEL
LIN {X 0,Y 587.344,Z 347.326,A -85,B 0,C 180,E1 -1297.839,E2 -1297.839} C_VEL
LIN {X 0,Y 587.321,Z 347.323,A -85,B 0,C 180,E1 -1300.254,E2 -1300.254} C_VEL
LIN {X 0,Y 587.318,Z 347.328,A -85,B 0,C 180,E1 -1303.118,E2 -1303.118} C_VEL
LIN {X 0,Y 587.34,Z 347.325,A -85,B 0,C 180,E1 -1306.051,E2 -1306.051} C_VEL
LIN {X 0,Y 587.34,Z 347.321,A -85,B 0,C 180,E1 -1308.925,E2 -1308.925} C_VEL
LIN {X 0,Y 587.332,Z 347.326,A -85,B 0,C 180,E1 -1311.521,E2 -1311.521} C_VEL
LIN {X 0,Y 587.294,Z 347.327,A -85,B 0,C 180,E1 -1314.1,E2 -1314.1} C_VEL
LIN {X 0,Y 587.34,Z 347.324,A -85,B 0,C 180,E1 -1316.603,E2 -1316.603} C_VEL
LIN {X 0,Y 587.339,Z 347.326,A -85,B 0,C 180,E1 -1319.49,E2 -1319.49} C_VEL
LIN {X 0,Y 587.356,Z 347.319,A -85,B 0,C 180,E1 -1322.307,E2 -1322.307} C_VEL
LIN {X 0,Y 587.338,Z 347.326,A -85,B 0,C 180,E1 -1324.483,E2 -1324.483} C_VEL
LIN {X 0,Y 587.344,Z 347.321,A -85,B 0,C 180,E1 -1327.486,E2 -1327.486} C_VEL
LIN {X 0,Y 587.318,Z 347.324,A -85,B 0,C 180,E1 -1330.424,E2 -1330.424} C_VEL
LIN {X 0,Y 587.352,Z 347.322,A -85,B 0,C 180,E1 -1333.311,E2 -1333.311} C_VEL
LIN {X 0,Y 587.362,Z 347.323,A -85,B 0,C 180,E1 -1336.154,E2 -1336.154} C_VEL
LIN {X 0,Y 587.346,Z 347.32,A -85,B 0,C 180,E1 -1338.962,E2 -1338.962} C_VEL
LIN {X 0,Y 587.37,Z 347.319,A -85,B 0,C 180,E1 -1341.745,E2 -1341.745} C_VEL
LIN {X 0,Y 587.369,Z 347.322,A -85,B 0,C 180,E1 -1344.507,E2 -1344.507} C_VEL
LIN {X 0,Y 587.372,Z 347.317,A -85,B 0,C 180,E1 -1347.257,E2 -1347.257} C_VEL
LIN {X 0,Y 587.388,Z 347.317,A -85,B 0,C 180,E1 -1350,E2 -1350} C_VEL
LIN {X 0,Y 587.372,Z 347.32,A -85,B 0,C 180,E1 -1352.743,E2 -1352.743} C_VEL
LIN {X 0,Y 587.363,Z 347.318,A -85,B 0,C 180,E1 -1355.493,E2 -1355.493} C_VEL
LIN {X 0,Y 587.369,Z 347.321,A -85,B 0,C 180,E1 -1358.255,E2 -1358.255} C_VEL
LIN {X 0,Y 587.353,Z 347.323,A -85,B 0,C 180,E1 -1361.134,E2 -1361.134} C_VEL
LIN {X 0,Y 587.37,Z 347.319,A -85,B 0,C 180,E1 -1364.26,E2 -1364.26} C_VEL
LIN {X 0,Y 587.36,Z 347.319,A -85,B 0,C 180,E1 -1367.406,E2 -1367.406} C_VEL
LIN {X 0,Y 587.33,Z 347.322,A -85,B 0,C 180,E1 -1370.305,E2 -1370.305} C_VEL
LIN {X 0,Y 587.325,Z 347.327,A -85,B 0,C 180,E1 -1373.259,E2 -1373.259} C_VEL
LIN {X 0,Y 587.339,Z 347.321,A -85,B 0,C 180,E1 -1375.516,E2 -1375.516} C_VEL
LIN {X 0,Y 587.353,Z 347.323,A -85,B 0,C 180,E1 -1377.818,E2 -1377.818} C_VEL
LIN {X 0,Y 587.338,Z 347.321,A -85,B 0,C 180,E1 -1380.509,E2 -1380.509} C_VEL
LIN {X 0,Y 587.339,Z 347.323,A -85,B 0,C 180,E1 -1383.396,E2 -1383.396} C_VEL
LIN {X 0,Y 587.294,Z 347.328,A -85,B 0,C 180,E1 -1385.9,E2 -1385.9} C_VEL
LIN {X 0,Y 587.335,Z 347.323,A -85,B 0,C 180,E1 -1388.479,E2 -1388.479} C_VEL
LIN {X 0,Y 587.338,Z 347.325,A -85,B 0,C 180,E1 -1391.157,E2 -1391.157} C_VEL
LIN {X 0,Y 587.33,Z 347.322,A -85,B 0,C 180,E1 -1394.113,E2 -1394.113} C_VEL
LIN {X 0,Y 587.316,Z 347.324,A -85,B 0,C 180,E1 -1396.993,E2 -1396.993} C_VEL
LIN {X 0,Y 587.316,Z 347.331,A -85,B 0,C 180,E1 -1399.745,E2 -1399.745} C_VEL
LIN {X 0,Y 587.346,Z 347.32,A -85,B 0,C 180,E1 -1402.392,E2 -1402.392} C_VEL
LIN {X 0,Y 587.366,Z 347.318,A -85,B 0,C 180,E1 -1405.78,E2 -1405.78} C_VEL
LIN {X 0,Y 587.341,Z 347.326,A -85,B 0,C 180,E1 -1408.231,E2 -1408.231} C_VEL
LIN {X 0,Y 587.353,Z 347.32,A -85,B 0,C 180,E1 -1410.867,E2 -1410.867} C_VEL
LIN {X 0,Y 587.34,Z 347.321,A -85,B 0,C 180,E1 -1413.721,E2 -1413.721} C_VEL
LIN {X 0,Y 587.34,Z 347.322,A -85,B 0,C 180,E1 -1415.994,E2 -1415.994} C_VEL
LIN {X 0,Y 587.323,Z 347.328,A -85,B 0,C 180,E1 -1418.226,E2 -1418.226} C_VEL
LIN {X 0,Y 587.355,Z 347.322,A -85,B 0,C 180,E1 -1421.151,E2 -1421.151} C_VEL
LIN {X 0,Y 587.325,Z 347.322,A -85,B 0,C 180,E1 -1424.025,E2 -1424.025} C_VEL
LIN {X 0,Y 587.362,Z 347.321,A -85,B 0,C 180,E1 -1426.154,E2 -1426.154} C_VEL
LIN {X 0,Y 587.342,Z 347.321,A -85,B 0,C 180,E1 -1428.962,E2 -1428.962} C_VEL
LIN {X 0,Y 587.372,Z 347.32,A -85,B 0,C 180,E1 -1431.745,E2 -1431.745} C_VEL
LIN {X 0,Y 587.362,Z 347.321,A -85,B 0,C 180,E1 -1434.507,E2 -1434.507} C_VEL
LIN {X 0,Y 587.376,Z 347.316,A -85,B 0,C 180,E1 -1437.257,E2 -1437.257} C_VEL
LIN {X 0,Y 587.387,Z 347.319,A -85,B 0,C 180,E1 -1440,E2 -1440} C_VEL
LIN {X 0,Y 587.381,Z 347.318,A -85,B 0,C 180,E1 -1442.743,E2 -1442.743} C_VEL
LIN {X 0,Y 587.357,Z 347.318,A -85,B 0,C 180,E1 -1445.493,E2 -1445.493} C_VEL
LIN {X 0,Y 587.344,Z 347.326,A -85,B 0,C 180,E1 -1448.256,E2 -1448.256} C_VEL
LIN {X 0,Y 587.352,Z 347.322,A -85,B 0,C 180,E1 -1451.134,E2 -1451.134} C_VEL
LIN {X 0,Y 587.368,Z 347.318,A -85,B 0,C 180,E1 -1454.26,E2 -1454.26} C_VEL
LIN {X 0,Y 587.351,Z 347.319,A -85,B 0,C 180,E1 -1457.406,E2 -1457.406} C_VEL
LIN {X 0,Y 587.33,Z 347.323,A -85,B 0,C 180,E1 -1460.305,E2 -1460.305} C_VEL
LIN {X 0,Y 587.317,Z 347.329,A -85,B 0,C 180,E1 -1463.259,E2 -1463.259} C_VEL
LIN {X 0,Y 587.334,Z 347.322,A -85,B 0,C 180,E1 -1465.517,E2 -1465.517} C_VEL
LIN {X 0,Y 587.349,Z 347.322,A -85,B 0,C 180,E1 -1467.818,E2 -1467.818} C_VEL
LIN {X 0,Y 587.342,Z 347.321,A -85,B 0,C 180,E1 -1470.51,E2 -1470.51} C_VEL
LIN {X 0,Y 587.337,Z 347.325,A -85,B 0,C 180,E1 -1473.397,E2 -1473.397} C_VEL
LIN {X 0,Y 587.323,Z 347.324,A -85,B 0,C 180,E1 -1475.898,E2 -1475.898} C_VEL
LIN {X 0,Y 587.337,Z 347.324,A -85,B 0,C 180,E1 -1478.479,E2 -1478.479} C_VEL
LIN {X 0,Y 587.338,Z 347.323,A -85,B 0,C 180,E1 -1481.157,E2 -1481.157} C_VEL
LIN {X 0,Y 587.337,Z 347.321,A -85,B 0,C 180,E1 -1484.114,E2 -1484.114} C_VEL
LIN {X 0,Y 587.325,Z 347.324,A -85,B 0,C 180,E1 -1486.994,E2 -1486.994} C_VEL
LIN {X 0,Y 587.315,Z 347.33,A -85,B 0,C 180,E1 -1489.746,E2 -1489.746} C_VEL
LIN {X 0,Y 587.346,Z 347.32,A -85,B 0,C 180,E1 -1492.392,E2 -1492.392} C_VEL
LIN {X 0,Y 587.364,Z 347.318,A -85,B 0,C 180,E1 -1495.78,E2 -1495.78} C_VEL
LIN {X 0,Y 587.347,Z 347.326,A -85,B 0,C 180,E1 -1498.231,E2 -1498.231} C_VEL
LIN {X 0,Y 587.353,Z 347.322,A -85,B 0,C 180,E1 -1500.867,E2 -1500.867} C_VEL
LIN {X 0,Y 587.351,Z 347.338,A -85,B 0,C 180,E1 -1501.745,E2 -1501.745} C_VEL
LIN {X 0,Y 588.037,Z 350.582,A -85,B 0,C 180,E1 -1502.332,E2 -1502.332} C_VEL
LIN {X 0,Y 587.882,Z 367.207,A -85,B 0,C 180,E1 -1505.077,E2 -1505.077} C_VEL
LIN {X 0,Y 587.742,Z 384.516,A -85,B 0,C 180,E1 -1507.873,E2 -1507.873} C_VEL
LIN {X 0,Y 587.618,Z 402.492,A -85,B 0,C 180,E1 -1510.721,E2 -1510.721} C_VEL
LIN {X 0,Y 587.486,Z 421.441,A -85,B 0,C 180,E1 -1513.673,E2 -1513.673} C_VEL
LIN {X 0,Y 587.399,Z 441.057,A -85,B 0,C 180,E1 -1516.684,E2 -1516.684} C_VEL
LIN {X 0,Y 587.364,Z 448.205,A -85,B 0,C 180,E1 -1517.749,E2 -1517.749} C_VEL
LIN {X 0,Y 587.727,Z 453.613,A -85,B 0,C 180,E1 -1517.833,E2 -1517.833} C_VEL
LIN {X 0,Y 587.69,Z 466.696,A -85,B 0,C 180,E1 -1518.117,E2 -1518.117} C_VEL
LIN {X 0,Y 587.639,Z 479.861,A -85,B 0,C 180,E1 -1518.556,E2 -1518.556} C_VEL
LIN {X 0,Y 587.532,Z 492.632,A -85,B 0,C 180,E1 -1519.141,E2 -1519.141} C_VEL
LIN {X 0,Y 587.467,Z 504.201,A -85,B 0,C 180,E1 -1519.837,E2 -1519.837} C_VEL
LIN {X 0,Y 587.367,Z 514.597,A -85,B 0,C 180,E1 -1520.617,E2 -1520.617} C_VEL
LIN {X 0,Y 587.321,Z 523.112,A -85,B 0,C 180,E1 -1521.398,E2 -1521.398} C_VEL
LIN {X 0,Y 587.274,Z 530.96,A -85,B 0,C 180,E1 -1522.263,E2 -1522.263} C_VEL
LIN {X 0,Y 587.23,Z 537.469,A -85,B 0,C 180,E1 -1523.126,E2 -1523.126} C_VEL
LIN {X 0,Y 587.236,Z 543.867,A -85,B 0,C 180,E1 -1524.161,E2 -1524.161} C_VEL
LIN {X 0,Y 587.147,Z 548.951,A -85,B 0,C 180,E1 -1525.194,E2 -1525.194} C_VEL
LIN {X 0,Y 587.212,Z 552.896,A -85,B 0,C 180,E1 -1526.226,E2 -1526.226} C_VEL
LIN {X 0,Y 587.132,Z 555.809,A -85,B 0,C 180,E1 -1527.256,E2 -1527.256} C_VEL
LIN {X 0,Y 587.141,Z 557.201,A -85,B 0,C 180,E1 -1527.942,E2 -1527.942} C_VEL
LIN {X 0,Y 587.14,Z 558.784,A -85,B 0,C 180,E1 -1529.314,E2 -1529.314} C_VEL
LIN {X 0,Y 587.137,Z 559,A -85,B 0,C 180,E1 -1530,E2 -1530} C_VEL
LIN {X 0,Y 587.147,Z 558.185,A -85,B 0,C 180,E1 -1531.372,E2 -1531.372} C_VEL
LIN {X 0,Y 587.141,Z 557.201,A -85,B 0,C 180,E1 -1532.058,E2 -1532.058} C_VEL
LIN {X 0,Y 587.132,Z 555.809,A -85,B 0,C 180,E1 -1532.744,E2 -1532.744} C_VEL
LIN {X 0,Y 587.212,Z 552.896,A -85,B 0,C 180,E1 -1533.774,E2 -1533.774} C_VEL
LIN {X 0,Y 587.147,Z 548.949,A -85,B 0,C 180,E1 -1534.806,E2 -1534.806} C_VEL
LIN {X 0,Y 587.217,Z 542.877,A -85,B 0,C 180,E1 -1536.011,E2 -1536.011} C_VEL
LIN {X 0,Y 587.245,Z 536.236,A -85,B 0,C 180,E1 -1537.046,E2 -1537.046} C_VEL
LIN {X 0,Y 587.299,Z 527.989,A -85,B 0,C 180,E1 -1538.083,E2 -1538.083} C_VEL
LIN {X 0,Y 587.343,Z 519.536,A -85,B 0,C 180,E1 -1538.949,E2 -1538.949} C_VEL
LIN {X 0,Y 587.422,Z 509.093,A -85,B 0,C 180,E1 -1539.816,E2 -1539.816} C_VEL
LIN {X 0,Y 587.488,Z 498.757,A -85,B 0,C 180,E1 -1540.512,E2 -1540.512} C_VEL
LIN {X 0,Y 587.583,Z 486.809,A -85,B 0,C 180,E1 -1541.149,E2 -1541.149} C_VEL
LIN {X 0,Y 587.63,Z 474.593,A -85,B 0,C 180,E1 -1541.639,E2 -1541.639} C_VEL
LIN {X 0,Y 587.679,Z 461.432,A -85,B 0,C 180,E1 -1542.015,E2 -1542.015} C_VEL
LIN {X 0,Y 587.517,Z 449.275,A -85,B 0,C 180,E1 -1542.234,E2 -1542.234} C_VEL
LIN {X 0,Y 587.347,Z 447.98,A -85,B 0,C 180,E1 -1542.263,E2 -1542.263} C_VEL
LIN {X 0,Y 587.452,Z 429.518,A -85,B 0,C 180,E1 -1545.082,E2 -1545.082} C_VEL
LIN {X 0,Y 587.541,Z 412.209,A -85,B 0,C 180,E1 -1547.76,E2 -1547.76} C_VEL
LIN {X 0,Y 587.657,Z 394.9,A -85,B 0,C 180,E1 -1550.476,E2 -1550.476} C_VEL
LIN {X 0,Y 587.781,Z 377.592,A -85,B 0,C 180,E1 -1553.24,E2 -1553.24} C_VEL
LIN {X 0,Y 587.964,Z 360.283,A -85,B 0,C 180,E1 -1556.058,E2 -1556.058} C_VEL
LIN {X 0,Y 587.881,Z 349.922,A -85,B 0,C 180,E1 -1557.79,E2 -1557.79} C_VEL
LIN {X 0,Y 587.363,Z 347.324,A -85,B 0,C 180,E1 -1558.303,E2 -1558.303} C_VEL
LIN {X 0,Y 587.333,Z 347.329,A -85,B 0,C 180,E1 -1560.967,E2 -1560.967} C_VEL
LIN {X 0,Y 587.34,Z 347.326,A -85,B 0,C 180,E1 -1563.397,E2 -1563.397} C_VEL
LIN {X 0,Y 587.294,Z 347.331,A -85,B 0,C 180,E1 -1565.9,E2 -1565.9} C_VEL
LIN {X 0,Y 587.324,Z 347.33,A -85,B 0,C 180,E1 -1568.48,E2 -1568.48} C_VEL
LIN {X 0,Y 587.34,Z 347.325,A -85,B 0,C 180,E1 -1571.157,E2 -1571.157} C_VEL
LIN {X 0,Y 587.338,Z 347.326,A -85,B 0,C 180,E1 -1574.114,E2 -1574.114} C_VEL
LIN {X 0,Y 587.325,Z 347.328,A -85,B 0,C 180,E1 -1576.994,E2 -1576.994} C_VEL
LIN {X 0,Y 587.322,Z 347.328,A -85,B 0,C 180,E1 -1579.746,E2 -1579.746} C_VEL
LIN {X 0,Y 587.347,Z 347.325,A -85,B 0,C 180,E1 -1582.392,E2 -1582.392} C_VEL
LIN {X 0,Y 587.333,Z 347.327,A -85,B 0,C 180,E1 -1584.945,E2 -1584.945} C_VEL
LIN {X 0,Y 587.342,Z 347.328,A -85,B 0,C 180,E1 -1587.421,E2 -1587.421} C_VEL
LIN {X 0,Y 587.365,Z 347.448,A -85,B 0,C 180,E1 -1590.326,E2 -1590.326} C_VEL
LIN {X 0,Y 587.326,Z 353.898,A -85,B 0,C 180,E1 -1592.954,E2 -1592.954} C_VEL
LIN {X 0,Y 587.296,Z 359.235,A -85,B 0,C 180,E1 -1595.239,E2 -1595.239} C_VEL
LIN {X 0,Y 587.245,Z 366.326,A -85,B 0,C 180,E1 -1598.223,E2 -1598.223} C_VEL
LIN {X 0,Y 587.243,Z 373.542,A -85,B 0,C 180,E1 -1601.148,E2 -1601.148} C_VEL
LIN {X 0,Y 587.221,Z 380.758,A -85,B 0,C 180,E1 -1604.022,E2 -1604.022} C_VEL
LIN {X 0,Y 587.177,Z 387.974,A -85,B 0,C 180,E1 -1606.855,E2 -1606.855} C_VEL
LIN {X 0,Y 587.137,Z 395.191,A -85,B 0,C 180,E1 -1609.657,E2 -1609.657} C_VEL
LIN {X 0,Y 587.145,Z 402.408,A -85,B 0,C 180,E1 -1612.434,E2 -1612.434} C_VEL
LIN {X 0,Y 587.173,Z 403.705,A -85,B 0,C 180,E1 -1612.931,E2 -1612.931} C_VEL
LIN {X 0,Y 587.346,Z 412.726,A -85,B 0,C 180,E1 -1613.238,E2 -1613.238} C_VEL
LIN {X 0,Y 587.308,Z 421.855,A -85,B 0,C 180,E1 -1613.693,E2 -1613.693} C_VEL
LIN {X 0,Y 587.248,Z 430.206,A -85,B 0,C 180,E1 -1614.248,E2 -1614.248} C_VEL
LIN {X 0,Y 587.216,Z 437.044,A -85,B 0,C 180,E1 -1614.85,E2 -1614.85} C_VEL
LIN {X 0,Y 587.216,Z 443.219,A -85,B 0,C 180,E1 -1615.538,E2 -1615.538} C_VEL
LIN {X 0,Y 587.227,Z 448.078,A -85,B 0,C 180,E1 -1616.226,E2 -1616.226} C_VEL
LIN {X 0,Y 587.183,Z 451.826,A -85,B 0,C 180,E1 -1616.913,E2 -1616.913} C_VEL
LIN {X 0,Y 587.145,Z 455.832,A -85,B 0,C 180,E1 -1617.942,E2 -1617.942} C_VEL
LIN {X 0,Y 587.147,Z 457.574,A -85,B 0,C 180,E1 -1618.628,E2 -1618.628} C_VEL
LIN {X 0,Y 587.141,Z 458.618,A -85,B 0,C 180,E1 -1619.314,E2 -1619.314} C_VEL
LIN {X 0,Y 587.137,Z 458.996,A -85,B 0,C 180,E1 -1620,E2 -1620} C_VEL
LIN {X 0,Y 587.14,Z 458.713,A -85,B 0,C 180,E1 -1620.686,E2 -1620.686} C_VEL
LIN {X 0,Y 587.149,Z 457.764,A -85,B 0,C 180,E1 -1621.372,E2 -1621.372} C_VEL
LIN {X 0,Y 587.144,Z 456.124,A -85,B 0,C 180,E1 -1622.058,E2 -1622.058} C_VEL
LIN {X 0,Y 587.145,Z 453.738,A -85,B 0,C 180,E1 -1622.744,E2 -1622.744} C_VEL
LIN {X 0,Y 587.228,Z 448.61,A -85,B 0,C 180,E1 -1623.774,E2 -1623.774} C_VEL
LIN {X 0,Y 587.247,Z 442.542,A -85,B 0,C 180,E1 -1624.634,E2 -1624.634} C_VEL
LIN {X 0,Y 587.197,Z 436.231,A -85,B 0,C 180,E1 -1625.322,E2 -1625.322} C_VEL
LIN {X 0,Y 587.249,Z 429.073,A -85,B 0,C 180,E1 -1625.925,E2 -1625.925} C_VEL
LIN {X 0,Y 587.28,Z 420.343,A -85,B 0,C 180,E1 -1626.484,E2 -1626.484} C_VEL
LIN {X 0,Y 587.368,Z 411.046,A -85,B 0,C 180,E1 -1626.915,E2 -1626.915} C_VEL
LIN {X 0,Y 587.161,Z 403.658,A -85,B 0,C 180,E1 -1627.177,E2 -1627.177} C_VEL
LIN {X 0,Y 587.176,Z 397.228,A -85,B 0,C 180,E1 -1629.647,E2 -1629.647} C_VEL
LIN {X 0,Y 587.166,Z 390.01,A -85,B 0,C 180,E1 -1632.442,E2 -1632.442} C_VEL
LIN {X 0,Y 587.186,Z 383.852,A -85,B 0,C 180,E1 -1634.849,E2 -1634.849} C_VEL
LIN {X 0,Y 587.22,Z 377.376,A -85,B 0,C 180,E1 -1637.41,E2 -1637.41} C_VEL
LIN {X 0,Y 587.198,Z 376.514,A -85,B 0,C 180,E1 -1637.754,E2 -1637.754} C_VEL
LIN {X 0,Y 586.526,Z 375.173,A -85,B 0,C 180,E1 -1638.312,E2 -1638.312} C_VEL
LIN {X 0,Y 583.675,Z 373.153,A -85,B 0,C 180,E1 -1639.22,E2 -1639.22} C_VEL
LIN {X 0,Y 581.272,Z 371.561,A -85,B 0,C 180,E1 -1639.951,E2 -1639.951} C_VEL
LIN {X 0,Y 580.244,Z 370.277,A -85,B 0,C 180,E1 -1640.514,E2 -1640.514} C_VEL
LIN {X 0,Y 580.162,Z 369.822,A -85,B 0,C 180,E1 -1640.704,E2 -1640.704} C_VEL
LIN {X 0,Y 580.207,Z 363.039,A -85,B 0,C 180,E1 -1643.561,E2 -1643.561} C_VEL
LIN {X 0,Y 580.281,Z 356.706,A -85,B 0,C 180,E1 -1646.331,E2 -1646.331} C_VEL
LIN {X 0,Y 580.335,Z 349.509,A -85,B 0,C 180,E1 -1649.315,E2 -1649.315} C_VEL
LIN {X 0,Y 580.341,Z 348.195,A -85,B 0,C 180,E1 -1649.97,E2 -1649.97} C_VEL
LIN {X 0,Y 580.293,Z 348.204,A -85,B 0,C 180,E1 -1653.025,E2 -1653.025} C_VEL
LIN {X 0,Y 580.282,Z 348.201,A -85,B 0,C 180,E1 -1655.761,E2 -1655.761} C_VEL
LIN {X 0,Y 580.293,Z 348.203,A -85,B 0,C 180,E1 -1658.146,E2 -1658.146} C_VEL
LIN {X 0,Y 580.303,Z 348.199,A -85,B 0,C 180,E1 -1660.843,E2 -1660.843} C_VEL
LIN {X 0,Y 580.276,Z 348.2,A -85,B 0,C 180,E1 -1663.658,E2 -1663.658} C_VEL
LIN {X 0,Y 580.29,Z 348.202,A -85,B 0,C 180,E1 -1666.608,E2 -1666.608} C_VEL
LIN {X 0,Y 580.302,Z 348.199,A -85,B 0,C 180,E1 -1669.157,E2 -1669.157} C_VEL
LIN {X 0,Y 580.293,Z 348.199,A -85,B 0,C 180,E1 -1671.927,E2 -1671.927} C_VEL
LIN {X 0,Y 580.254,Z 348.208,A -85,B 0,C 180,E1 -1674.453,E2 -1674.453} C_VEL
LIN {X 0,Y 580.296,Z 348.198,A -85,B 0,C 180,E1 -1676.975,E2 -1676.975} C_VEL
LIN {X 0,Y 580.299,Z 348.202,A -85,B 0,C 180,E1 -1679.425,E2 -1679.425} C_VEL
LIN {X 0,Y 580.303,Z 348.197,A -85,B 0,C 180,E1 -1682.141,E2 -1682.141} C_VEL
LIN {X 0,Y 580.326,Z 348.194,A -85,B 0,C 180,E1 -1685.27,E2 -1685.27} C_VEL
LIN {X 0,Y 580.278,Z 348.207,A -85,B 0,C 180,E1 -1687.947,E2 -1687.947} C_VEL
LIN {X 0,Y 580.302,Z 348.2,A -85,B 0,C 180,E1 -1690.913,E2 -1690.913} C_VEL
LIN {X 0,Y 580.279,Z 348.2,A -85,B 0,C 180,E1 -1693.825,E2 -1693.825} C_VEL
LIN {X 0,Y 580.33,Z 348.197,A -85,B 0,C 180,E1 -1695.983,E2 -1695.983} C_VEL
LIN {X 0,Y 580.31,Z 348.196,A -85,B 0,C 180,E1 -1698.827,E2 -1698.827} C_VEL
LIN {X 0,Y 580.333,Z 348.197,A -85,B 0,C 180,E1 -1701.644,E2 -1701.644} C_VEL
LIN {X 0,Y 580.336,Z 348.198,A -85,B 0,C 180,E1 -1704.44,E2 -1704.44} C_VEL
LIN {X 0,Y 580.346,Z 348.198,A -85,B 0,C 180,E1 -1707.918,E2 -1707.918} C_VEL
LIN {X 0,Y 580.362,Z 348.19,A -85,B 0,C 180,E1 -1710.694,E2 -1710.694} C_VEL
LIN {X 0,Y 580.285,Z 348.201,A -85,B 0,C 180,E1 -1713.472,E2 -1713.472} C_VEL
LIN {X 0,Y 580.331,Z 348.194,A -85,B 0,C 180,E1 -1715.56,E2 -1715.56} C_VEL
LIN {X 0,Y 580.331,Z 348.196,A -85,B 0,C 180,E1 -1718.356,E2 -1718.356} C_VEL
LIN {X 0,Y 580.305,Z 348.202,A -85,B 0,C 180,E1 -1721.191,E2 -1721.191} C_VEL
LIN {X 0,Y 580.33,Z 348.194,A -85,B 0,C 180,E1 -1724.017,E2 -1724.017} C_VEL
LIN {X 0,Y 580.317,Z 348.196,A -85,B 0,C 180,E1 -1726.914,E2 -1726.914} C_VEL
LIN {X 0,Y 580.306,Z 348.202,A -85,B 0,C 180,E1 -1729.822,E2 -1729.822} C_VEL
LIN {X 0,Y 580.299,Z 348.202,A -85,B 0,C 180,E1 -1732.802,E2 -1732.802} C_VEL
LIN {X 0,Y 580.311,Z 348.199,A -85,B 0,C 180,E1 -1735.08,E2 -1735.08} C_VEL
LIN {X 0,Y 580.305,Z 348.202,A -85,B 0,C 180,E1 -1738.185,E2 -1738.185} C_VEL
LIN {X 0,Y 580.286,Z 348.199,A -85,B 0,C 180,E1 -1740.694,E2 -1740.694} C_VEL
LIN {X 0,Y 580.309,Z 348.2,A -85,B 0,C 180,E1 -1743.316,E2 -1743.316} C_VEL
LIN {X 0,Y 580.25,Z 348.205,A -85,B 0,C 180,E1 -1745.756,E2 -1745.756} C_VEL
LIN {X 0,Y 580.293,Z 348.205,A -85,B 0,C 180,E1 -1748.146,E2 -1748.146} C_VEL
LIN {X 0,Y 580.302,Z 348.198,A -85,B 0,C 180,E1 -1750.843,E2 -1750.843} C_VEL
LIN {X 0,Y 580.283,Z 348.2,A -85,B 0,C 180,E1 -1753.658,E2 -1753.658} C_VEL
LIN {X 0,Y 580.277,Z 348.205,A -85,B 0,C 180,E1 -1756.61,E2 -1756.61} C_VEL
LIN {X 0,Y 580.3,Z 348.199,A -85,B 0,C 180,E1 -1759.156,E2 -1759.156} C_VEL
LIN {X 0,Y 580.292,Z 348.199,A -85,B 0,C 180,E1 -1761.927,E2 -1761.927} C_VEL
LIN {X 0,Y 580.256,Z 348.206,A -85,B 0,C 180,E1 -1764.453,E2 -1764.453} C_VEL
LIN {X 0,Y 580.293,Z 348.199,A -85,B 0,C 180,E1 -1766.975,E2 -1766.975} C_VEL
LIN {X 0,Y 580.3,Z 348.201,A -85,B 0,C 180,E1 -1769.425,E2 -1769.425} C_VEL
LIN {X 0,Y 580.301,Z 348.198,A -85,B 0,C 180,E1 -1772.141,E2 -1772.141} C_VEL
LIN {X 0,Y 580.325,Z 348.196,A -85,B 0,C 180,E1 -1775.27,E2 -1775.27} C_VEL
LIN {X 0,Y 580.275,Z 348.206,A -85,B 0,C 180,E1 -1777.947,E2 -1777.947} C_VEL
LIN {X 0,Y 580.323,Z 348.196,A -85,B 0,C 180,E1 -1780.914,E2 -1780.914} C_VEL
LIN {X 0,Y 580.279,Z 348.2,A -85,B 0,C 180,E1 -1783.825,E2 -1783.825} C_VEL
LIN {X 0,Y 580.329,Z 348.195,A -85,B 0,C 180,E1 -1785.983,E2 -1785.983} C_VEL
LIN {X 0,Y 580.308,Z 348.197,A -85,B 0,C 180,E1 -1788.827,E2 -1788.827} C_VEL
LIN {X 0,Y 580.336,Z 348.198,A -85,B 0,C 180,E1 -1791.644,E2 -1791.644} C_VEL
LIN {X 0,Y 580.327,Z 348.197,A -85,B 0,C 180,E1 -1794.44,E2 -1794.44} C_VEL
LIN {X 0,Y 580.343,Z 348.192,A -85,B 0,C 180,E1 -1797.223,E2 -1797.223} C_VEL
LIN {X 0,Y 580.356,Z 348.195,A -85,B 0,C 180,E1 -1800,E2 -1800} C_VEL
LIN {X 0,Y 580.347,Z 348.195,A -85,B 0,C 180,E1 -1802.776,E2 -1802.776} C_VEL
LIN {X 0,Y 580.323,Z 348.195,A -85,B 0,C 180,E1 -1805.56,E2 -1805.56} C_VEL
LIN {X 0,Y 580.326,Z 348.196,A -85,B 0,C 180,E1 -1807.655,E2 -1807.655} C_VEL
LIN {X 0,Y 580.304,Z 348.198,A -85,B 0,C 180,E1 -1810.467,E2 -1810.467} C_VEL
LIN {X 0,Y 580.279,Z 348.205,A -85,B 0,C 180,E1 -1813.304,E2 -1813.304} C_VEL
LIN {X 0,Y 580.298,Z 348.198,A -85,B 0,C 180,E1 -1815.453,E2 -1815.453} C_VEL
LIN {X 0,Y 580.293,Z 348.199,A -85,B 0,C 180,E1 -1817.625,E2 -1817.625} C_VEL
LIN {X 0,Y 580.307,Z 348.204,A -85,B 0,C 180,E1 -1819.822,E2 -1819.822} C_VEL
LIN {X 0,Y 580.293,Z 348.201,A -85,B 0,C 180,E1 -1822.803,E2 -1822.803} C_VEL
LIN {X 0,Y 580.309,Z 348.2,A -85,B 0,C 180,E1 -1825.08,E2 -1825.08} C_VEL
LIN {X 0,Y 580.301,Z 348.204,A -85,B 0,C 180,E1 -1828.186,E2 -1828.186} C_VEL
LIN {X 0,Y 580.291,Z 348.199,A -85,B 0,C 180,E1 -1830.695,E2 -1830.695} C_VEL
LIN {X 0,Y 580.306,Z 348.202,A -85,B 0,C 180,E1 -1833.316,E2 -1833.316} C_VEL
LIN {X 0,Y 580.28,Z 348.2,A -85,B 0,C 180,E1 -1835.761,E2 -1835.761} C_VEL
LIN {X 0,Y 580.293,Z 348.206,A -85,B 0,C 180,E1 -1838.146,E2 -1838.146} C_VEL
LIN {X 0,Y 580.3,Z 348.198,A -85,B 0,C 180,E1 -1840.843,E2 -1840.843} C_VEL
LIN {X 0,Y 580.291,Z 348.2,A -85,B 0,C 180,E1 -1843.657,E2 -1843.657} C_VEL
LIN {X 0,Y 580.288,Z 348.205,A -85,B 0,C 180,E1 -1846.608,E2 -1846.608} C_VEL
LIN {X 0,Y 580.301,Z 348.198,A -85,B 0,C 180,E1 -1849.157,E2 -1849.157} C_VEL
LIN {X 0,Y 580.291,Z 348.2,A -85,B 0,C 180,E1 -1851.927,E2 -1851.927} C_VEL
LIN {X 0,Y 580.255,Z 348.206,A -85,B 0,C 180,E1 -1854.453,E2 -1854.453} C_VEL
LIN {X 0,Y 580.295,Z 348.199,A -85,B 0,C 180,E1 -1856.975,E2 -1856.975} C_VEL
LIN {X 0,Y 580.299,Z 348.2,A -85,B 0,C 180,E1 -1859.425,E2 -1859.425} C_VEL
LIN {X 0,Y 580.316,Z 348.276,A -85,B 0,C 180,E1 -1861.52,E2 -1861.52} C_VEL
LIN {X 0,Y 581.177,Z 352.795,A -85,B 0,C 180,E1 -1862.342,E2 -1862.342} C_VEL
LIN {X 0,Y 580.986,Z 368.361,A -85,B 0,C 180,E1 -1864.952,E2 -1864.952} C_VEL
LIN {X 0,Y 580.811,Z 385.67,A -85,B 0,C 180,E1 -1867.782,E2 -1867.782} C_VEL
LIN {X 0,Y 580.641,Z 404.203,A -85,B 0,C 180,E1 -1870.753,E2 -1870.753} C_VEL
LIN {X 0,Y 580.497,Z 422.595,A -85,B 0,C 180,E1 -1873.651,E2 -1873.651} C_VEL
LIN {X 0,Y 580.368,Z 441.057,A -85,B 0,C 180,E1 -1876.52,E2 -1876.52} C_VEL
LIN {X 0,Y 580.328,Z 448.205,A -85,B 0,C 180,E1 -1877.598,E2 -1877.598} C_VEL
LIN {X 0,Y 580.799,Z 453.612,A -85,B 0,C 180,E1 -1877.686,E2 -1877.686} C_VEL
LIN {X 0,Y 580.764,Z 466.696,A -85,B 0,C 180,E1 -1877.973,E2 -1877.973} C_VEL
LIN {X 0,Y 580.672,Z 479.174,A -85,B 0,C 180,E1 -1878.389,E2 -1878.389} C_VEL
LIN {X 0,Y 580.585,Z 490.928,A -85,B 0,C 180,E1 -1878.921,E2 -1878.921} C_VEL
LIN {X 0,Y 580.479,Z 501.583,A -85,B 0,C 180,E1 -1879.537,E2 -1879.537} C_VEL
LIN {X 0,Y 580.38,Z 512.474,A -85,B 0,C 180,E1 -1880.327,E2 -1880.327} C_VEL
LIN {X 0,Y 580.271,Z 523.112,A -85,B 0,C 180,E1 -1881.292,E2 -1881.292} C_VEL
LIN {X 0,Y 580.222,Z 530.96,A -85,B 0,C 180,E1 -1882.168,E2 -1882.168} C_VEL
LIN {X 0,Y 580.154,Z 538.651,A -85,B 0,C 180,E1 -1883.222,E2 -1883.222} C_VEL
LIN {X 0,Y 580.139,Z 545.68,A -85,B 0,C 180,E1 -1884.439,E2 -1884.439} C_VEL
LIN {X 0,Y 580.108,Z 550.371,A -85,B 0,C 180,E1 -1885.483,E2 -1885.483} C_VEL
LIN {X 0,Y 580.123,Z 553.956,A -85,B 0,C 180,E1 -1886.527,E2 -1886.527} C_VEL
LIN {X 0,Y 580.043,Z 555.808,A -85,B 0,C 180,E1 -1887.222,E2 -1887.222} C_VEL
LIN {X 0,Y 580.04,Z 557.2,A -85,B 0,C 180,E1 -1887.917,E2 -1887.917} C_VEL
LIN {X 0,Y 580.04,Z 558.784,A -85,B 0,C 180,E1 -1889.306,E2 -1889.306} C_VEL
LIN {X 0,Y 580.037,Z 559,A -85,B 0,C 180,E1 -1890,E2 -1890} C_VEL
LIN {X 0,Y 580.047,Z 558.185,A -85,B 0,C 180,E1 -1891.389,E2 -1891.389} C_VEL
LIN {X 0,Y 580.04,Z 557.2,A -85,B 0,C 180,E1 -1892.083,E2 -1892.083} C_VEL
LIN {X 0,Y 580.043,Z 555.81,A -85,B 0,C 180,E1 -1892.778,E2 -1892.778} C_VEL
LIN {X 0,Y 580.109,Z 552.896,A -85,B 0,C 180,E1 -1893.821,E2 -1893.821} C_VEL
LIN {X 0,Y 580.053,Z 548.949,A -85,B 0,C 180,E1 -1894.865,E2 -1894.865} C_VEL
LIN {X 0,Y 580.139,Z 542.877,A -85,B 0,C 180,E1 -1896.085,E2 -1896.085} C_VEL
LIN {X 0,Y 580.184,Z 536.236,A -85,B 0,C 180,E1 -1897.132,E2 -1897.132} C_VEL
LIN {X 0,Y 580.25,Z 527.989,A -85,B 0,C 180,E1 -1898.182,E2 -1898.182} C_VEL
LIN {X 0,Y 580.308,Z 519.537,A -85,B 0,C 180,E1 -1899.058,E2 -1899.058} C_VEL
LIN {X 0,Y 580.425,Z 509.095,A -85,B 0,C 180,E1 -1899.936,E2 -1899.936} C_VEL
LIN {X 0,Y 580.494,Z 498.755,A -85,B 0,C 180,E1 -1900.64,E2 -1900.64} C_VEL
LIN {X 0,Y 580.597,Z 487.24,A -85,B 0,C 180,E1 -1901.264,E2 -1901.264} C_VEL
LIN {X 0,Y 580.685,Z 474.468,A -85,B 0,C 180,E1 -1901.785,E2 -1901.785} C_VEL
LIN {X 0,Y 580.76,Z 461.431,A -85,B 0,C 180,E1 -1902.16,E2 -1902.16} C_VEL
LIN {X 0,Y 580.616,Z 450.218,A -85,B 0,C 180,E1 -1902.368,E2 -1902.368} C_VEL
LIN {X 0,Y 580.314,Z 447.98,A -85,B 0,C 180,E1 -1902.414,E2 -1902.414} C_VEL
LIN {X 0,Y 580.438,Z 430.672,A -85,B 0,C 180,E1 -1905.089,E2 -1905.089} C_VEL
LIN {X 0,Y 580.544,Z 413.363,A -85,B 0,C 180,E1 -1907.799,E2 -1907.799} C_VEL
LIN {X 0,Y 580.698,Z 396.054,A -85,B 0,C 180,E1 -1910.547,E2 -1910.547} C_VEL
LIN {X 0,Y 580.86,Z 379.127,A -85,B 0,C 180,E1 -1913.282,E2 -1913.282} C_VEL
LIN {X 0,Y 581.102,Z 361.608,A -85,B 0,C 180,E1 -1916.167,E2 -1916.167} C_VEL
LIN {X 0,Y 581.208,Z 352.862,A -85,B 0,C 180,E1 -1917.659,E2 -1917.659} C_VEL
LIN {X 0,Y 580.299,Z 348.204,A -85,B 0,C 180,E1 -1918.531,E2 -1918.531} C_VEL
LIN {X 0,Y 580.281,Z 348.205,A -85,B 0,C 180,E1 -1921.385,E2 -1921.385} C_VEL
LIN {X 0,Y 580.32,Z 348.201,A -85,B 0,C 180,E1 -1923.855,E2 -1923.855} C_VEL
LIN {X 0,Y 580.301,Z 348.203,A -85,B 0,C 180,E1 -1926.934,E2 -1926.934} C_VEL
LIN {X 0,Y 580.287,Z 348.204,A -85,B 0,C 180,E1 -1929.934,E2 -1929.934} C_VEL
LIN {X 0,Y 580.285,Z 348.206,A -85,B 0,C 180,E1 -1932.706,E2 -1932.706} C_VEL
LIN {X 0,Y 580.278,Z 348.206,A -85,B 0,C 180,E1 -1935.609,E2 -1935.609} C_VEL
LIN {X 0,Y 580.318,Z 348.2,A -85,B 0,C 180,E1 -1938.234,E2 -1938.234} C_VEL
LIN {X 0,Y 580.293,Z 348.205,A -85,B 0,C 180,E1 -1940.966,E2 -1940.966} C_VEL
LIN {X 0,Y 580.275,Z 348.206,A -85,B 0,C 180,E1 -1943.597,E2 -1943.597} C_VEL
LIN {X 0,Y 580.321,Z 348.201,A -85,B 0,C 180,E1 -1946.145,E2 -1946.145} C_VEL
LIN {X 0,Y 580.281,Z 348.206,A -85,B 0,C 180,E1 -1948.615,E2 -1948.615} C_VEL
LIN {X 0,Y 580.311,Z 348.32,A -85,B 0,C 180,E1 -1950.294,E2 -1950.294} C_VEL
LIN {X 0,Y 580.263,Z 355.802,A -85,B 0,C 180,E1 -1953.376,E2 -1953.376} C_VEL
LIN {X 0,Y 580.232,Z 361.212,A -85,B 0,C 180,E1 -1955.681,E2 -1955.681} C_VEL
LIN {X 0,Y 580.198,Z 366.328,A -85,B 0,C 180,E1 -1957.944,E2 -1957.944} C_VEL
LIN {X 0,Y 580.184,Z 373.544,A -85,B 0,C 180,E1 -1960.909,E2 -1960.909} C_VEL
LIN {X 0,Y 580.148,Z 380.76,A -85,B 0,C 180,E1 -1963.822,E2 -1963.822} C_VEL
LIN {X 0,Y 580.09,Z 387.976,A -85,B 0,C 180,E1 -1966.692,E2 -1966.692} C_VEL
LIN {X 0,Y 580.057,Z 395.193,A -85,B 0,C 180,E1 -1969.529,E2 -1969.529} C_VEL
LIN {X 0,Y 580.068,Z 402.409,A -85,B 0,C 180,E1 -1972.341,E2 -1972.341} C_VEL
LIN {X 0,Y 580.073,Z 403.706,A -85,B 0,C 180,E1 -1972.844,E2 -1972.844} C_VEL
LIN {X 0,Y 580.304,Z 411.831,A -85,B 0,C 180,E1 -1973.119,E2 -1973.119} C_VEL
LIN {X 0,Y 580.255,Z 420.748,A -85,B 0,C 180,E1 -1973.551,E2 -1973.551} C_VEL
LIN {X 0,Y 580.188,Z 429.031,A -85,B 0,C 180,E1 -1974.09,E2 -1974.09} C_VEL
LIN {X 0,Y 580.144,Z 437.048,A -85,B 0,C 180,E1 -1974.787,E2 -1974.787} C_VEL
LIN {X 0,Y 580.151,Z 443.223,A -85,B 0,C 180,E1 -1975.484,E2 -1975.484} C_VEL
LIN {X 0,Y 580.157,Z 448.081,A -85,B 0,C 180,E1 -1976.18,E2 -1976.18} C_VEL
LIN {X 0,Y 580.095,Z 451.828,A -85,B 0,C 180,E1 -1976.875,E2 -1976.875} C_VEL
LIN {X 0,Y 580.047,Z 455.835,A -85,B 0,C 180,E1 -1977.917,E2 -1977.917} C_VEL
LIN {X 0,Y 580.047,Z 457.576,A -85,B 0,C 180,E1 -1978.611,E2 -1978.611} C_VEL
LIN {X 0,Y 580.042,Z 458.619,A -85,B 0,C 180,E1 -1979.306,E2 -1979.306} C_VEL
LIN {X 0,Y 580.038,Z 458.996,A -85,B 0,C 180,E1 -1980,E2 -1980} C_VEL
LIN {X 0,Y 580.04,Z 458.712,A -85,B 0,C 180,E1 -1980.694,E2 -1980.694} C_VEL
LIN {X 0,Y 580.049,Z 457.763,A -85,B 0,C 180,E1 -1981.389,E2 -1981.389} C_VEL
LIN {X 0,Y 580.046,Z 456.122,A -85,B 0,C 180,E1 -1982.083,E2 -1982.083} C_VEL
LIN {X 0,Y 580.057,Z 453.736,A -85,B 0,C 180,E1 -1982.778,E2 -1982.778} C_VEL
LIN {X 0,Y 580.158,Z 448.607,A -85,B 0,C 180,E1 -1983.82,E2 -1983.82} C_VEL
LIN {X 0,Y 580.182,Z 442.538,A -85,B 0,C 180,E1 -1984.69,E2 -1984.69} C_VEL
LIN {X 0,Y 580.121,Z 436.225,A -85,B 0,C 180,E1 -1985.387,E2 -1985.387} C_VEL
LIN {X 0,Y 580.202,Z 429.067,A -85,B 0,C 180,E1 -1985.997,E2 -1985.997} C_VEL
LIN {X 0,Y 580.232,Z 421.325,A -85,B 0,C 180,E1 -1986.505,E2 -1986.505} C_VEL
LIN {X 0,Y 580.334,Z 412.204,A -85,B 0,C 180,E1 -1986.956,E2 -1986.956} C_VEL
LIN {X 0,Y 580.058,Z 403.656,A -85,B 0,C 180,E1 -1987.265,E2 -1987.265} C_VEL
LIN {X 0,Y 580.076,Z 397.227,A -85,B 0,C 180,E1 -1989.766,E2 -1989.766} C_VEL
LIN {X 0,Y 580.084,Z 390.008,A -85,B 0,C 180,E1 -1992.596,E2 -1992.596} C_VEL
LIN {X 0,Y 580.125,Z 384.594,A -85,B 0,C 180,E1 -1994.739,E2 -1994.739} C_VEL
LIN {X 0,Y 580.148,Z 377.374,A -85,B 0,C 180,E1 -1997.629,E2 -1997.629} C_VEL
LIN {X 0,Y 580.16,Z 371.96,A -85,B 0,C 180,E1 -1999.828,E2 -1999.828} C_VEL
LIN {X 0,Y 580.162,Z 369.822,A -85,B 0,C 180,E1 -2000.704,E2 -2000.704} C_VEL
LIN {X 0,Y 579.495,Z 368.529,A -85,B 0,C 180,E1 -2001.269,E2 -2001.269} C_VEL
LIN {X 0,Y 576.634,Z 366.665,A -85,B 0,C 180,E1 -2002.191,E2 -2002.191} C_VEL
LIN {X 0,Y 574.232,Z 365.221,A -85,B 0,C 180,E1 -2002.934,E2 -2002.934} C_VEL
LIN {X 0,Y 573.224,Z 364.037,A -85,B 0,C 180,E1 -2003.506,E2 -2003.506} C_VEL
LIN {X 0,Y 573.154,Z 363.61,A -85,B 0,C 180,E1 -2003.699,E2 -2003.699} C_VEL
LIN {X 0,Y 573.231,Z 357.882,A -85,B 0,C 180,E1 -2006.192,E2 -2006.192} C_VEL
LIN {X 0,Y 573.298,Z 349.998,A -85,B 0,C 180,E1 -2009.497,E2 -2009.497} C_VEL
LIN {X 0,Y 573.313,Z 349.071,A -85,B 0,C 180,E1 -2009.985,E2 -2009.985} C_VEL
LIN {X 0,Y 573.257,Z 349.078,A -85,B 0,C 180,E1 -2012.645,E2 -2012.645} C_VEL
LIN {X 0,Y 573.26,Z 349.075,A -85,B 0,C 180,E1 -2015.184,E2 -2015.184} C_VEL
LIN {X 0,Y 573.24,Z 349.083,A -85,B 0,C 180,E1 -2017.807,E2 -2017.807} C_VEL
LIN {X 0,Y 573.274,Z 349.073,A -85,B 0,C 180,E1 -2020.528,E2 -2020.528} C_VEL
LIN {X 0,Y 573.242,Z 349.076,A -85,B 0,C 180,E1 -2023.668,E2 -2023.668} C_VEL
LIN {X 0,Y 573.251,Z 349.078,A -85,B 0,C 180,E1 -2026.642,E2 -2026.642} C_VEL
LIN {X 0,Y 573.248,Z 349.082,A -85,B 0,C 180,E1 -2029.475,E2 -2029.475} C_VEL
LIN {X 0,Y 573.239,Z 349.077,A -85,B 0,C 180,E1 -2032.192,E2 -2032.192} C_VEL
LIN {X 0,Y 573.239,Z 349.078,A -85,B 0,C 180,E1 -2035.229,E2 -2035.229} C_VEL
LIN {X 0,Y 573.257,Z 349.08,A -85,B 0,C 180,E1 -2037.772,E2 -2037.772} C_VEL
LIN {X 0,Y 573.269,Z 349.074,A -85,B 0,C 180,E1 -2040.634,E2 -2040.634} C_VEL
LIN {X 0,Y 573.256,Z 349.081,A -85,B 0,C 180,E1 -2043.024,E2 -2043.024} C_VEL
LIN {X 0,Y 573.279,Z 349.072,A -85,B 0,C 180,E1 -2045.366,E2 -2045.366} C_VEL
LIN {X 0,Y 573.234,Z 349.08,A -85,B 0,C 180,E1 -2048.419,E2 -2048.419} C_VEL
LIN {X 0,Y 573.274,Z 349.074,A -85,B 0,C 180,E1 -2050.731,E2 -2050.731} C_VEL
LIN {X 0,Y 573.252,Z 349.076,A -85,B 0,C 180,E1 -2053.622,E2 -2053.622} C_VEL
LIN {X 0,Y 573.277,Z 349.073,A -85,B 0,C 180,E1 -2055.807,E2 -2055.807} C_VEL
LIN {X 0,Y 573.268,Z 349.074,A -85,B 0,C 180,E1 -2058.745,E2 -2058.745} C_VEL
LIN {X 0,Y 573.289,Z 349.075,A -85,B 0,C 180,E1 -2061.54,E2 -2061.54} C_VEL
LIN {X 0,Y 573.303,Z 349.073,A -85,B 0,C 180,E1 -2064.372,E2 -2064.372} C_VEL
LIN {X 0,Y 573.316,Z 349.073,A -85,B 0,C 180,E1 -2067.892,E2 -2067.892} C_VEL
LIN {X 0,Y 573.333,Z 349.066,A -85,B 0,C 180,E1 -2070.702,E2 -2070.702} C_VEL
LIN {X 0,Y 573.306,Z 349.074,A -85,B 0,C 180,E1 -2072.811,E2 -2072.811} C_VEL
LIN {X 0,Y 573.298,Z 349.07,A -85,B 0,C 180,E1 -2075.628,E2 -2075.628} C_VEL
LIN {X 0,Y 573.287,Z 349.072,A -85,B 0,C 180,E1 -2078.459,E2 -2078.459} C_VEL
LIN {X 0,Y 573.277,Z 349.079,A -85,B 0,C 180,E1 -2081.312,E2 -2081.312} C_VEL
LIN {X 0,Y 573.286,Z 349.075,A -85,B 0,C 180,E1 -2084.424,E2 -2084.424} C_VEL
LIN {X 0,Y 573.264,Z 349.074,A -85,B 0,C 180,E1 -2087.111,E2 -2087.111} C_VEL
LIN {X 0,Y 573.254,Z 349.077,A -85,B 0,C 180,E1 -2090.077,E2 -2090.077} C_VEL
LIN {X 0,Y 573.239,Z 349.084,A -85,B 0,C 180,E1 -2093.099,E2 -2093.099} C_VEL
LIN {X 0,Y 573.259,Z 349.075,A -85,B 0,C 180,E1 -2095.41,E2 -2095.41} C_VEL
LIN {X 0,Y 573.258,Z 349.082,A -85,B 0,C 180,E1 -2098.029,E2 -2098.029} C_VEL
LIN {X 0,Y 573.231,Z 349.079,A -85,B 0,C 180,E1 -2100.882,E2 -2100.882} C_VEL
LIN {X 0,Y 573.266,Z 349.075,A -85,B 0,C 180,E1 -2103.524,E2 -2103.524} C_VEL
LIN {X 0,Y 573.218,Z 349.083,A -85,B 0,C 180,E1 -2106.051,E2 -2106.051} C_VEL
LIN {X 0,Y 573.252,Z 349.076,A -85,B 0,C 180,E1 -2108.701,E2 -2108.701} C_VEL
LIN {X 0,Y 573.234,Z 349.082,A -85,B 0,C 180,E1 -2111.593,E2 -2111.593} C_VEL
LIN {X 0,Y 573.239,Z 349.079,A -85,B 0,C 180,E1 -2114.333,E2 -2114.333} C_VEL
LIN {X 0,Y 573.243,Z 349.077,A -85,B 0,C 180,E1 -2117.358,E2 -2117.358} C_VEL
LIN {X 0,Y 573.244,Z 349.077,A -85,B 0,C 180,E1 -2120.392,E2 -2120.392} C_VEL
LIN {X 0,Y 573.255,Z 349.082,A -85,B 0,C 180,E1 -2123.077,E2 -2123.077} C_VEL
LIN {X 0,Y 573.272,Z 349.073,A -85,B 0,C 180,E1 -2125.671,E2 -2125.671} C_VEL
LIN {X 0,Y 573.242,Z 349.083,A -85,B 0,C 180,E1 -2128.184,E2 -2128.184} C_VEL
LIN {X 0,Y 573.268,Z 349.074,A -85,B 0,C 180,E1 -2130.634,E2 -2130.634} C_VEL
LIN {X 0,Y 573.253,Z 349.082,A -85,B 0,C 180,E1 -2133.024,E2 -2133.024} C_VEL
LIN {X 0,Y 573.278,Z 349.073,A -85,B 0,C 180,E1 -2135.366,E2 -2135.366} C_VEL
LIN {X 0,Y 573.232,Z 349.081,A -85,B 0,C 180,E1 -2138.419,E2 -2138.419} C_VEL
LIN {X 0,Y 573.282,Z 349.072,A -85,B 0,C 180,E1 -2140.728,E2 -2140.728} C_VEL
LIN {X 0,Y 573.251,Z 349.076,A -85,B 0,C 180,E1 -2143.622,E2 -2143.622} C_VEL
LIN {X 0,Y 573.276,Z 349.073,A -85,B 0,C 180,E1 -2145.807,E2 -2145.807} C_VEL
LIN {X 0,Y 573.266,Z 349.074,A -85,B 0,C 180,E1 -2148.745,E2 -2148.745} C_VEL
LIN {X 0,Y 573.293,Z 349.077,A -85,B 0,C 180,E1 -2151.541,E2 -2151.541} C_VEL
LIN {X 0,Y 573.294,Z 349.072,A -85,B 0,C 180,E1 -2154.372,E2 -2154.372} C_VEL
LIN {X 0,Y 573.312,Z 349.072,A -85,B 0,C 180,E1 -2157.892,E2 -2157.892} C_VEL
LIN {X 0,Y 573.335,Z 349.066,A -85,B 0,C 180,E1 -2160.702,E2 -2160.702} C_VEL
LIN {X 0,Y 573.242,Z 349.079,A -85,B 0,C 180,E1 -2163.514,E2 -2163.514} C_VEL
LIN {X 0,Y 573.291,Z 349.071,A -85,B 0,C 180,E1 -2165.628,E2 -2165.628} C_VEL
LIN {X 0,Y 573.274,Z 349.075,A -85,B 0,C 180,E1 -2167.75,E2 -2167.75} C_VEL
LIN {X 0,Y 573.27,Z 349.074,A -85,B 0,C 180,E1 -2170.597,E2 -2170.597} C_VEL
LIN {X 0,Y 573.269,Z 349.076,A -85,B 0,C 180,E1 -2172.748,E2 -2172.748} C_VEL
LIN {X 0,Y 573.239,Z 349.083,A -85,B 0,C 180,E1 -2174.92,E2 -2174.92} C_VEL
LIN {X 0,Y 573.261,Z 349.075,A -85,B 0,C 180,E1 -2177.112,E2 -2177.112} C_VEL
LIN {X 0,Y 573.254,Z 349.079,A -85,B 0,C 180,E1 -2180.077,E2 -2180.077} C_VEL
LIN {X 0,Y 573.237,Z 349.084,A -85,B 0,C 180,E1 -2183.099,E2 -2183.099} C_VEL
LIN {X 0,Y 573.256,Z 349.076,A -85,B 0,C 180,E1 -2185.41,E2 -2185.41} C_VEL
LIN {X 0,Y 573.253,Z 349.081,A -85,B 0,C 180,E1 -2188.029,E2 -2188.029} C_VEL
LIN {X 0,Y 573.236,Z 349.078,A -85,B 0,C 180,E1 -2190.883,E2 -2190.883} C_VEL
LIN {X 0,Y 573.265,Z 349.077,A -85,B 0,C 180,E1 -2193.524,E2 -2193.524} C_VEL
LIN {X 0,Y 573.248,Z 349.078,A -85,B 0,C 180,E1 -2196.049,E2 -2196.049} C_VEL
LIN {X 0,Y 573.25,Z 349.077,A -85,B 0,C 180,E1 -2198.701,E2 -2198.701} C_VEL
LIN {X 0,Y 573.233,Z 349.084,A -85,B 0,C 180,E1 -2201.593,E2 -2201.593} C_VEL
LIN {X 0,Y 573.243,Z 349.078,A -85,B 0,C 180,E1 -2204.333,E2 -2204.333} C_VEL
LIN {X 0,Y 573.246,Z 349.077,A -85,B 0,C 180,E1 -2207.358,E2 -2207.358} C_VEL
LIN {X 0,Y 573.241,Z 349.077,A -85,B 0,C 180,E1 -2210.392,E2 -2210.392} C_VEL
LIN {X 0,Y 573.255,Z 349.081,A -85,B 0,C 180,E1 -2213.078,E2 -2213.078} C_VEL
LIN {X 0,Y 573.271,Z 349.073,A -85,B 0,C 180,E1 -2215.671,E2 -2215.671} C_VEL
LIN {X 0,Y 573.246,Z 349.081,A -85,B 0,C 180,E1 -2218.185,E2 -2218.185} C_VEL
LIN {X 0,Y 573.288,Z 349.142,A -85,B 0,C 180,E1 -2221.276,E2 -2221.276} C_VEL
LIN {X 0,Y 574.334,Z 354.638,A -85,B 0,C 180,E1 -2222.29,E2 -2222.29} C_VEL
LIN {X 0,Y 574.093,Z 368.383,A -85,B 0,C 180,E1 -2224.63,E2 -2224.63} C_VEL
LIN {X 0,Y 573.874,Z 385.67,A -85,B 0,C 180,E1 -2227.499,E2 -2227.499} C_VEL
LIN {X 0,Y 573.658,Z 402.981,A -85,B 0,C 180,E1 -2230.312,E2 -2230.312} C_VEL
LIN {X 0,Y 573.521,Z 421.553,A -85,B 0,C 180,E1 -2233.281,E2 -2233.281} C_VEL
LIN {X 0,Y 573.349,Z 439.904,A -85,B 0,C 180,E1 -2236.171,E2 -2236.171} C_VEL
LIN {X 0,Y 573.279,Z 448.092,A -85,B 0,C 180,E1 -2237.442,E2 -2237.442} C_VEL
LIN {X 0,Y 573.88,Z 453.612,A -85,B 0,C 180,E1 -2237.535,E2 -2237.535} C_VEL
LIN {X 0,Y 573.831,Z 466.695,A -85,B 0,C 180,E1 -2237.826,E2 -2237.826} C_VEL
LIN {X 0,Y 573.719,Z 479.916,A -85,B 0,C 180,E1 -2238.276,E2 -2238.276} C_VEL
LIN {X 0,Y 573.591,Z 492.63,A -85,B 0,C 180,E1 -2238.873,E2 -2238.873} C_VEL
LIN {X 0,Y 573.434,Z 504.202,A -85,B 0,C 180,E1 -2239.585,E2 -2239.585} C_VEL
LIN {X 0,Y 573.334,Z 514.599,A -85,B 0,C 180,E1 -2240.386,E2 -2240.386} C_VEL
LIN {X 0,Y 573.241,Z 523.112,A -85,B 0,C 180,E1 -2241.185,E2 -2241.185} C_VEL
LIN {X 0,Y 573.161,Z 530.96,A -85,B 0,C 180,E1 -2242.071,E2 -2242.071} C_VEL
LIN {X 0,Y 573.073,Z 538.581,A -85,B 0,C 180,E1 -2243.126,E2 -2243.126} C_VEL
LIN {X 0,Y 573.07,Z 545.68,A -85,B 0,C 180,E1 -2244.37,E2 -2244.37} C_VEL
LIN {X 0,Y 573.028,Z 550.371,A -85,B 0,C 180,E1 -2245.428,E2 -2245.428} C_VEL
LIN {X 0,Y 573.022,Z 553.957,A -85,B 0,C 180,E1 -2246.484,E2 -2246.484} C_VEL
LIN {X 0,Y 572.959,Z 555.808,A -85,B 0,C 180,E1 -2247.188,E2 -2247.188} C_VEL
LIN {X 0,Y 572.939,Z 557.199,A -85,B 0,C 180,E1 -2247.891,E2 -2247.891} C_VEL
LIN {X 0,Y 572.94,Z 558.785,A -85,B 0,C 180,E1 -2249.297,E2 -2249.297} C_VEL
LIN {X 0,Y 572.938,Z 559,A -85,B 0,C 180,E1 -2250,E2 -2250} C_VEL
LIN {X 0,Y 572.946,Z 558.186,A -85,B 0,C 180,E1 -2251.406,E2 -2251.406} C_VEL
LIN {X 0,Y 572.939,Z 557.2,A -85,B 0,C 180,E1 -2252.109,E2 -2252.109} C_VEL
LIN {X 0,Y 572.959,Z 555.81,A -85,B 0,C 180,E1 -2252.812,E2 -2252.812} C_VEL
LIN {X 0,Y 573.014,Z 552.896,A -85,B 0,C 180,E1 -2253.868,E2 -2253.868} C_VEL
LIN {X 0,Y 572.963,Z 548.949,A -85,B 0,C 180,E1 -2254.926,E2 -2254.926} C_VEL
LIN {X 0,Y 573.064,Z 542.876,A -85,B 0,C 180,E1 -2256.16,E2 -2256.16} C_VEL
LIN {X 0,Y 573.119,Z 536.237,A -85,B 0,C 180,E1 -2257.221,E2 -2257.221} C_VEL
LIN {X 0,Y 573.201,Z 527.99,A -85,B 0,C 180,E1 -2258.283,E2 -2258.283} C_VEL
LIN {X 0,Y 573.287,Z 519.537,A -85,B 0,C 180,E1 -2259.17,E2 -2259.17} C_VEL
LIN {X 0,Y 573.43,Z 509.096,A -85,B 0,C 180,E1 -2260.058,E2 -2260.058} C_VEL
LIN {X 0,Y 573.51,Z 498.773,A -85,B 0,C 180,E1 -2260.77,E2 -2260.77} C_VEL
LIN {X 0,Y 573.629,Z 487.586,A -85,B 0,C 180,E1 -2261.386,E2 -2261.386} C_VEL
LIN {X 0,Y 573.729,Z 475.764,A -85,B 0,C 180,E1 -2261.885,E2 -2261.885} C_VEL
LIN {X 0,Y 573.815,Z 462.344,A -85,B 0,C 180,E1 -2262.287,E2 -2262.287} C_VEL
LIN {X 0,Y 573.714,Z 451.064,A -85,B 0,C 180,E1 -2262.507,E2 -2262.507} C_VEL
LIN {X 0,Y 573.261,Z 447.98,A -85,B 0,C 180,E1 -2262.569,E2 -2262.569} C_VEL
LIN {X 0,Y 573.408,Z 430.672,A -85,B 0,C 180,E1 -2265.279,E2 -2265.279} C_VEL
LIN {X 0,Y 573.551,Z 414.517,A -85,B 0,C 180,E1 -2267.839,E2 -2267.839} C_VEL
LIN {X 0,Y 573.757,Z 397.208,A -85,B 0,C 180,E1 -2270.62,E2 -2270.62} C_VEL
LIN {X 0,Y 573.954,Z 380.742,A -85,B 0,C 180,E1 -2273.311,E2 -2273.311} C_VEL
LIN {X 0,Y 574.216,Z 363.877,A -85,B 0,C 180,E1 -2276.143,E2 -2276.143} C_VEL
LIN {X 0,Y 574.394,Z 354.809,A -85,B 0,C 180,E1 -2277.707,E2 -2277.707} C_VEL
LIN {X 0,Y 573.27,Z 349.08,A -85,B 0,C 180,E1 -2278.813,E2 -2278.813} C_VEL
LIN {X 0,Y 573.246,Z 349.082,A -85,B 0,C 180,E1 -2281.815,E2 -2281.815} C_VEL
LIN {X 0,Y 573.271,Z 349.08,A -85,B 0,C 180,E1 -2284.329,E2 -2284.329} C_VEL
LIN {X 0,Y 573.254,Z 349.082,A -85,B 0,C 180,E1 -2287.166,E2 -2287.166} C_VEL
LIN {X 0,Y 573.241,Z 349.083,A -85,B 0,C 180,E1 -2289.608,E2 -2289.608} C_VEL
LIN {X 0,Y 573.247,Z 349.083,A -85,B 0,C 180,E1 -2292.642,E2 -2292.642} C_VEL
LIN {X 0,Y 573.243,Z 349.083,A -85,B 0,C 180,E1 -2295.667,E2 -2295.667} C_VEL
LIN {X 0,Y 573.248,Z 349.081,A -85,B 0,C 180,E1 -2298.544,E2 -2298.544} C_VEL
LIN {X 0,Y 573.252,Z 349.081,A -85,B 0,C 180,E1 -2301.299,E2 -2301.299} C_VEL
LIN {X 0,Y 573.242,Z 349.083,A -85,B 0,C 180,E1 -2304.015,E2 -2304.015} C_VEL
LIN {X 0,Y 573.289,Z 349.077,A -85,B 0,C 180,E1 -2306.519,E2 -2306.519} C_VEL
LIN {X 0,Y 573.233,Z 349.084,A -85,B 0,C 180,E1 -2309.118,E2 -2309.118} C_VEL
LIN {X 0,Y 573.28,Z 349.279,A -85,B 0,C 180,E1 -2310.292,E2 -2310.292} C_VEL
LIN {X 0,Y 573.204,Z 355.799,A -85,B 0,C 180,E1 -2313.022,E2 -2313.022} C_VEL
LIN {X 0,Y 573.227,Z 361.502,A -85,B 0,C 180,E1 -2315.364,E2 -2315.364} C_VEL
LIN {X 0,Y 573.167,Z 366.571,A -85,B 0,C 180,E1 -2317.659,E2 -2317.659} C_VEL
LIN {X 0,Y 573.078,Z 371.741,A -85,B 0,C 180,E1 -2319.917,E2 -2319.917} C_VEL
LIN {X 0,Y 573.086,Z 379.363,A -85,B 0,C 180,E1 -2323.049,E2 -2323.049} C_VEL
LIN {X 0,Y 573.05,Z 386.173,A -85,B 0,C 180,E1 -2325.801,E2 -2325.801} C_VEL
LIN {X 0,Y 573.015,Z 393.868,A -85,B 0,C 180,E1 -2328.873,E2 -2328.873} C_VEL
LIN {X 0,Y 572.986,Z 400.607,A -85,B 0,C 180,E1 -2331.536,E2 -2331.536} C_VEL
LIN {X 0,Y 572.969,Z 403.708,A -85,B 0,C 180,E1 -2332.755,E2 -2332.755} C_VEL
LIN {X 0,Y 573.264,Z 411.917,A -85,B 0,C 180,E1 -2333.037,E2 -2333.037} C_VEL
LIN {X 0,Y 573.185,Z 420.756,A -85,B 0,C 180,E1 -2333.471,E2 -2333.471} C_VEL
LIN {X 0,Y 573.139,Z 429.04,A -85,B 0,C 180,E1 -2334.017,E2 -2334.017} C_VEL
LIN {X 0,Y 573.054,Z 437.053,A -85,B 0,C 180,E1 -2334.722,E2 -2334.722} C_VEL
LIN {X 0,Y 573.089,Z 443.227,A -85,B 0,C 180,E1 -2335.428,E2 -2335.428} C_VEL
LIN {X 0,Y 573.089,Z 448.085,A -85,B 0,C 180,E1 -2336.133,E2 -2336.133} C_VEL
LIN {X 0,Y 573.012,Z 451.831,A -85,B 0,C 180,E1 -2336.836,E2 -2336.836} C_VEL
LIN {X 0,Y 572.951,Z 455.837,A -85,B 0,C 180,E1 -2337.891,E2 -2337.891} C_VEL
LIN {X 0,Y 572.947,Z 457.578,A -85,B 0,C 180,E1 -2338.594,E2 -2338.594} C_VEL
LIN {X 0,Y 572.942,Z 458.62,A -85,B 0,C 180,E1 -2339.297,E2 -2339.297} C_VEL
LIN {X 0,Y 572.938,Z 458.996,A -85,B 0,C 180,E1 -2340,E2 -2340} C_VEL
LIN {X 0,Y 572.941,Z 458.711,A -85,B 0,C 180,E1 -2340.703,E2 -2340.703} C_VEL
LIN {X 0,Y 572.949,Z 457.762,A -85,B 0,C 180,E1 -2341.406,E2 -2341.406} C_VEL
LIN {X 0,Y 572.95,Z 456.12,A -85,B 0,C 180,E1 -2342.109,E2 -2342.109} C_VEL
LIN {X 0,Y 572.973,Z 453.733,A -85,B 0,C 180,E1 -2342.812,E2 -2342.812} C_VEL
LIN {X 0,Y 573.085,Z 448.604,A -85,B 0,C 180,E1 -2343.868,E2 -2343.868} C_VEL
LIN {X 0,Y 573.111,Z 442.532,A -85,B 0,C 180,E1 -2344.748,E2 -2344.748} C_VEL
LIN {X 0,Y 573.05,Z 436.219,A -85,B 0,C 180,E1 -2345.454,E2 -2345.454} C_VEL
LIN {X 0,Y 573.156,Z 429.061,A -85,B 0,C 180,E1 -2346.071,E2 -2346.071} C_VEL
LIN {X 0,Y 573.196,Z 421.314,A -85,B 0,C 180,E1 -2346.586,E2 -2346.586} C_VEL
LIN {X 0,Y 573.298,Z 412.19,A -85,B 0,C 180,E1 -2347.042,E2 -2347.042} C_VEL
LIN {X 0,Y 572.974,Z 403.655,A -85,B 0,C 180,E1 -2347.356,E2 -2347.356} C_VEL
LIN {X 0,Y 572.988,Z 397.226,A -85,B 0,C 180,E1 -2349.888,E2 -2349.888} C_VEL
LIN {X 0,Y 573.01,Z 391.811,A -85,B 0,C 180,E1 -2352.035,E2 -2352.035} C_VEL
LIN {X 0,Y 573.049,Z 384.592,A -85,B 0,C 180,E1 -2354.925,E2 -2354.925} C_VEL
LIN {X 0,Y 573.084,Z 377.373,A -85,B 0,C 180,E1 -2357.854,E2 -2357.854} C_VEL
LIN {X 0,Y 573.108,Z 370.164,A -85,B 0,C 180,E1 -2360.832,E2 -2360.832} C_VEL
LIN {X 0,Y 573.154,Z 363.61,A -85,B 0,C 180,E1 -2363.699,E2 -2363.699} C_VEL
LIN {X 0,Y 572.53,Z 362.414,A -85,B 0,C 180,E1 -2364.273,E2 -2364.273} C_VEL
LIN {X 0,Y 569.726,Z 360.669,A -85,B 0,C 180,E1 -2365.209,E2 -2365.209} C_VEL
LIN {X 0,Y 567.323,Z 359.157,A -85,B 0,C 180,E1 -2365.962,E2 -2365.962} C_VEL
LIN {X 0,Y 566.274,Z 357.878,A -85,B 0,C 180,E1 -2366.54,E2 -2366.54} C_VEL
LIN {X 0,Y 566.179,Z 357.423,A -85,B 0,C 180,E1 -2366.735,E2 -2366.735} C_VEL
LIN {X 0,Y 566.266,Z 349.949,A -85,B 0,C 180,E1 -2369.97,E2 -2369.97} C_VEL
LIN {X 0,Y 566.224,Z 349.956,A -85,B 0,C 180,E1 -2373.102,E2 -2373.102} C_VEL
LIN {X 0,Y 566.201,Z 349.955,A -85,B 0,C 180,E1 -2375.69,E2 -2375.69} C_VEL
LIN {X 0,Y 566.22,Z 349.953,A -85,B 0,C 180,E1 -2378.559,E2 -2378.559} C_VEL
LIN {X 0,Y 566.207,Z 349.959,A -85,B 0,C 180,E1 -2381.137,E2 -2381.137} C_VEL
LIN {X 0,Y 566.196,Z 349.955,A -85,B 0,C 180,E1 -2384.036,E2 -2384.036} C_VEL
LIN {X 0,Y 566.209,Z 349.953,A -85,B 0,C 180,E1 -2387.082,E2 -2387.082} C_VEL
LIN {X 0,Y 566.211,Z 349.958,A -85,B 0,C 180,E1 -2389.801,E2 -2389.801} C_VEL
LIN {X 0,Y 566.203,Z 349.956,A -85,B 0,C 180,E1 -2392.599,E2 -2392.599} C_VEL
LIN {X 0,Y 566.202,Z 349.954,A -85,B 0,C 180,E1 -2395.181,E2 -2395.181} C_VEL
